LIN {X 0,Y 163.912,Z 823.88,A -85,B 0,C 180,E1 24592.6,E2 24592.6} C_VEL
LIN {X 0,Y 165.468,Z 824.667,A -85,B 0,C 180,E1 24598.513,E2 24598.513} C_VEL
LIN {X 0,Y 168.195,Z 823.745,A -85,B 0,C 180,E1 24603.972,E2 24603.972} C_VEL
LIN {X 0,Y 172.518,Z 820.86,A -85,B 0,C 180,E1 24609.607,E2 24609.607} C_VEL
LIN {X 0,Y 177.878,Z 816.328,A -85,B 0,C 180,E1 24614.638,E2 24614.638} C_VEL
LIN {X 0,Y 183.953,Z 810.223,A -85,B 0,C 180,E1 24619.07,E2 24619.07} C_VEL
LIN {X 0,Y 190.994,Z 802.117,A -85,B 0,C 180,E1 24623.221,E2 24623.221} C_VEL
LIN {X 0,Y 197.72,Z 793.266,A -85,B 0,C 180,E1 24626.552,E2 24626.552} C_VEL
LIN {X 0,Y 204.701,Z 782.624,A -85,B 0,C 180,E1 24629.553,E2 24629.553} C_VEL
LIN {X 0,Y 211.875,Z 769.936,A -85,B 0,C 180,E1 24632.25,E2 24632.25} C_VEL
LIN {X 0,Y 217.985,Z 757.04,A -85,B 0,C 180,E1 24634.33,E2 24634.33} C_VEL
LIN {X 0,Y 223.609,Z 742.371,A -85,B 0,C 180,E1 24636.121,E2 24636.121} C_VEL
LIN {X 0,Y 228.283,Z 726.827,A -85,B 0,C 180,E1 24637.541,E2 24637.541} C_VEL
LIN {X 0,Y 231.741,Z 710.644,A -85,B 0,C 180,E1 24638.599,E2 24638.599} C_VEL
LIN {X 0,Y 234.04,Z 693.375,A -85,B 0,C 180,E1 24639.347,E2 24639.347} C_VEL
LIN {X 0,Y 240.538,Z 622.169,A -85,B 0,C 180,E1 24641.299,E2 24641.299} C_VEL
LIN {X 0,Y 239.787,Z 607.797,A -85,B 0,C 180,E1 24642.742,E2 24642.742} C_VEL
LIN {X 0,Y 236.069,Z 599.284,A -85,B 0,C 180,E1 24645.591,E2 24645.591} C_VEL
LIN {X 0,Y 232.297,Z 591.41,A -85,B 0,C 180,E1 24649.02,E2 24649.02} C_VEL
LIN {X 0,Y 229.336,Z 585.624,A -85,B 0,C 180,E1 24652.358,E2 24652.358} C_VEL
LIN {X 0,Y 226.439,Z 580.103,A -85,B 0,C 180,E1 24656.962,E2 24656.962} C_VEL
LIN {X 0,Y 225.491,Z 578.392,A -85,B 0,C 180,E1 24659.237,E2 24659.237} C_VEL
LIN {X 0,Y 224.567,Z 575.979,A -85,B 0,C 180,E1 24664.596,E2 24664.596} C_VEL
LIN {X 0,Y 224.605,Z 575.941,A -85,B 0,C 180,E1 24665.938,E2 24665.938} C_VEL
LIN {X 0,Y 224.734,Z 577.003,A -85,B 0,C 180,E1 24667.755,E2 24667.755} C_VEL
LIN {X 0,Y 224.996,Z 580.824,A -85,B 0,C 180,E1 24670.283,E2 24670.283} C_VEL
LIN {X 0,Y 225.974,Z 586.453,A -85,B 0,C 180,E1 24673.585,E2 24673.585} C_VEL
LIN {X 0,Y 226.496,Z 587.496,A -85,B 0,C 180,E1 24674.544,E2 24674.544} C_VEL
LIN {X 0,Y 228.557,Z 590.668,A -85,B 0,C 180,E1 24677.509,E2 24677.509} C_VEL
LIN {X 0,Y 230.127,Z 593.107,A -85,B 0,C 180,E1 24679.347,E2 24679.347} C_VEL
LIN {X 0,Y 233.43,Z 598.617,A -85,B 0,C 180,E1 24682.541,E2 24682.541} C_VEL
LIN {X 0,Y 236.72,Z 604.703,A -85,B 0,C 180,E1 24685.252,E2 24685.252} C_VEL
LIN {X 0,Y 239.579,Z 610.555,A -85,B 0,C 180,E1 24687.307,E2 24687.307} C_VEL
LIN {X 0,Y 229.729,Z 717.254,A -85,B 0,C 180,E1 24690.022,E2 24690.022} C_VEL
LIN {X 0,Y 226.439,Z 735.292,A -85,B 0,C 180,E1 24690.738,E2 24690.738} C_VEL
LIN {X 0,Y 222.025,Z 751.667,A -85,B 0,C 180,E1 24691.665,E2 24691.665} C_VEL
LIN {X 0,Y 216.24,Z 768.025,A -85,B 0,C 180,E1 24692.942,E2 24692.942} C_VEL
LIN {X 0,Y 209.368,Z 783.676,A -85,B 0,C 180,E1 24694.631,E2 24694.631} C_VEL
LIN {X 0,Y 201.664,Z 798.456,A -85,B 0,C 180,E1 24696.802,E2 24696.802} C_VEL
LIN {X 0,Y 193.264,Z 812.488,A -85,B 0,C 180,E1 24699.57,E2 24699.57} C_VEL
LIN {X 0,Y 184.592,Z 825.393,A -85,B 0,C 180,E1 24703.01,E2 24703.01} C_VEL
LIN {X 0,Y 176.218,Z 836.632,A -85,B 0,C 180,E1 24707.088,E2 24707.088} C_VEL
LIN {X 0,Y 168.557,Z 846.394,A -85,B 0,C 180,E1 24711.909,E2 24711.909} C_VEL
LIN {X 0,Y 161.973,Z 854.666,A -85,B 0,C 180,E1 24717.518,E2 24717.518} C_VEL
LIN {X 0,Y 156.956,Z 861.39,A -85,B 0,C 180,E1 24723.925,E2 24723.925} C_VEL
LIN {X 0,Y 154.079,Z 866.16,A -85,B 0,C 180,E1 24730.674,E2 24730.674} C_VEL
LIN {X 0,Y 153.336,Z 869.27,A -85,B 0,C 180,E1 24737.986,E2 24737.986} C_VEL
LIN {X 0,Y 154.463,Z 870.381,A -85,B 0,C 180,E1 24744.801,E2 24744.801} C_VEL
LIN {X 0,Y 155.627,Z 870.068,A -85,B 0,C 180,E1 24749.264,E2 24749.264} C_VEL
LIN {X 0,Y 155.435,Z 869.168,A -85,B 0,C 180,E1 24752.213,E2 24752.213} C_VEL
LIN {X 0,Y 154.206,Z 866.135,A -85,B 0,C 180,E1 24757.826,E2 24757.826} C_VEL
LIN {X 0,Y 153.721,Z 861.161,A -85,B 0,C 180,E1 24763.926,E2 24763.926} C_VEL
LIN {X 0,Y 154.617,Z 854.342,A -85,B 0,C 180,E1 24770.044,E2 24770.044} C_VEL
LIN {X 0,Y 157.051,Z 845.493,A -85,B 0,C 180,E1 24776.059,E2 24776.059} C_VEL
LIN {X 0,Y 160.791,Z 835.076,A -85,B 0,C 180,E1 24781.49,E2 24781.49} C_VEL
LIN {X 0,Y 165.105,Z 824.003,A -85,B 0,C 180,E1 24785.975,E2 24785.975} C_VEL
LIN {X 0,Y 170.211,Z 811.051,A -85,B 0,C 180,E1 24790.034,E2 24790.034} C_VEL
LIN {X 0,Y 175.619,Z 796.472,A -85,B 0,C 180,E1 24793.544,E2 24793.544} C_VEL
LIN {X 0,Y 180.883,Z 780.858,A -85,B 0,C 180,E1 24796.397,E2 24796.397} C_VEL
LIN {X 0,Y 185.452,Z 765.246,A -85,B 0,C 180,E1 24798.54,E2 24798.54} C_VEL
LIN {X 0,Y 189.399,Z 748.752,A -85,B 0,C 180,E1 24800.199,E2 24800.199} C_VEL
LIN {X 0,Y 192.481,Z 731.114,A -85,B 0,C 180,E1 24801.451,E2 24801.451} C_VEL
LIN {X 0,Y 194.415,Z 712.665,A -85,B 0,C 180,E1 24802.3,E2 24802.3} C_VEL
LIN {X 0,Y 202.526,Z 587.616,A -85,B 0,C 180,E1 24806.166,E2 24806.166} C_VEL
LIN {X 0,Y 202.127,Z 580.747,A -85,B 0,C 180,E1 24806.612,E2 24806.612} C_VEL
LIN {X 0,Y 194.488,Z 565.099,A -85,B 0,C 180,E1 24809.663,E2 24809.663} C_VEL
LIN {X 0,Y 186.875,Z 551.393,A -85,B 0,C 180,E1 24813.036,E2 24813.036} C_VEL
LIN {X 0,Y 183.387,Z 545.505,A -85,B 0,C 180,E1 24814.833,E2 24814.833} C_VEL
LIN {X 0,Y 180.867,Z 537.663,A -85,B 0,C 180,E1 24819.281,E2 24819.281} C_VEL
LIN {X 0,Y 178.385,Z 530.763,A -85,B 0,C 180,E1 24824.06,E2 24824.06} C_VEL
LIN {X 0,Y 176.409,Z 525.313,A -85,B 0,C 180,E1 24828.559,E2 24828.559} C_VEL
LIN {X 0,Y 174.729,Z 521.276,A -85,B 0,C 180,E1 24832.768,E2 24832.768} C_VEL
LIN {X 0,Y 173.264,Z 517.729,A -85,B 0,C 180,E1 24837.355,E2 24837.355} C_VEL
LIN {X 0,Y 171.645,Z 513.857,A -85,B 0,C 180,E1 24845.013,E2 24845.013} C_VEL
LIN {X 0,Y 170.767,Z 512.763,A -85,B 0,C 180,E1 24851.484,E2 24851.484} C_VEL
LIN {X 0,Y 170.898,Z 512.989,A -85,B 0,C 180,E1 24858.065,E2 24858.065} C_VEL
LIN {X 0,Y 171.446,Z 514.088,A -85,B 0,C 180,E1 24862.639,E2 24862.639} C_VEL
LIN {X 0,Y 172.787,Z 517.698,A -85,B 0,C 180,E1 24869.846,E2 24869.846} C_VEL
LIN {X 0,Y 174.086,Z 521.491,A -85,B 0,C 180,E1 24874.782,E2 24874.782} C_VEL
LIN {X 0,Y 175.487,Z 525.746,A -85,B 0,C 180,E1 24879.205,E2 24879.205} C_VEL
LIN {X 0,Y 177.274,Z 531.253,A -85,B 0,C 180,E1 24883.928,E2 24883.928} C_VEL
LIN {X 0,Y 179.348,Z 538.517,A -85,B 0,C 180,E1 24889.062,E2 24889.062} C_VEL
LIN {X 0,Y 181.315,Z 546.515,A -85,B 0,C 180,E1 24893.839,E2 24893.839} C_VEL
LIN {X 0,Y 182.26,Z 550.218,A -85,B 0,C 180,E1 24895.653,E2 24895.653} C_VEL
LIN {X 0,Y 188.742,Z 562.541,A -85,B 0,C 180,E1 24898.821,E2 24898.821} C_VEL
LIN {X 0,Y 194.269,Z 574.356,A -85,B 0,C 180,E1 24901.293,E2 24901.293} C_VEL
LIN {X 0,Y 197.448,Z 613.753,A -85,B 0,C 180,E1 24904.282,E2 24904.282} C_VEL
LIN {X 0,Y 191.617,Z 696.457,A -85,B 0,C 180,E1 24907.072,E2 24907.072} C_VEL
LIN {X 0,Y 189.522,Z 713.957,A -85,B 0,C 180,E1 24908.201,E2 24908.201} C_VEL
LIN {X 0,Y 186.823,Z 729.138,A -85,B 0,C 180,E1 24909.642,E2 24909.642} C_VEL
LIN {X 0,Y 183.113,Z 744.763,A -85,B 0,C 180,E1 24911.701,E2 24911.701} C_VEL
LIN {X 0,Y 178.862,Z 759.406,A -85,B 0,C 180,E1 24914.268,E2 24914.268} C_VEL
LIN {X 0,Y 174.27,Z 772.863,A -85,B 0,C 180,E1 24917.407,E2 24917.407} C_VEL
LIN {X 0,Y 169.559,Z 785.286,A -85,B 0,C 180,E1 24921.18,E2 24921.18} C_VEL
LIN {X 0,Y 165.156,Z 796.018,A -85,B 0,C 180,E1 24925.485,E2 24925.485} C_VEL
LIN {X 0,Y 161.321,Z 805.271,A -85,B 0,C 180,E1 24930.354,E2 24930.354} C_VEL
LIN {X 0,Y 158.455,Z 812.493,A -85,B 0,C 180,E1 24935.431,E2 24935.431} C_VEL
LIN {X 0,Y 156.409,Z 818.667,A -85,B 0,C 180,E1 24941.429,E2 24941.429} C_VEL
LIN {X 0,Y 155.668,Z 822.689,A -85,B 0,C 180,E1 24947.184,E2 24947.184} C_VEL
LIN {X 0,Y 156.104,Z 825.148,A -85,B 0,C 180,E1 24953.397,E2 24953.397} C_VEL
LIN {X 0,Y 157.914,Z 825.868,A -85,B 0,C 180,E1 24959.595,E2 24959.595} C_VEL
LIN {X 0,Y 161.208,Z 824.71,A -85,B 0,C 180,E1 24965.662,E2 24965.662} C_VEL
LIN {X 0,Y 166.048,Z 821.661,A -85,B 0,C 180,E1 24971.48,E2 24971.48} C_VEL
LIN {X 0,Y 171.989,Z 816.833,A -85,B 0,C 180,E1 24976.685,E2 24976.685} C_VEL
LIN {X 0,Y 179.003,Z 810.086,A -85,B 0,C 180,E1 24981.443,E2 24981.443} C_VEL
LIN {X 0,Y 186.039,Z 802.321,A -85,B 0,C 180,E1 24985.314,E2 24985.314} C_VEL
LIN {X 0,Y 193.796,Z 792.352,A -85,B 0,C 180,E1 24988.919,E2 24988.919} C_VEL
LIN {X 0,Y 201.556,Z 780.804,A -85,B 0,C 180,E1 24992.006,E2 24992.006} C_VEL
LIN {X 0,Y 208.433,Z 768.711,A -85,B 0,C 180,E1 24994.422,E2 24994.422} C_VEL
LIN {X 0,Y 215.191,Z 754.374,A -85,B 0,C 180,E1 24996.585,E2 24996.585} C_VEL
LIN {X 0,Y 220.706,Z 739.879,A -85,B 0,C 180,E1 24998.233,E2 24998.233} C_VEL
LIN {X 0,Y 225.369,Z 723.672,A -85,B 0,C 180,E1 24999.588,E2 24999.588} C_VEL
LIN {X 0,Y 228.761,Z 706.983,A -85,B 0,C 180,E1 25000.578,E2 25000.578} C_VEL
LIN {X 0,Y 230.892,Z 688.612,A -85,B 0,C 180,E1 25001.264,E2 25001.264} C_VEL
LIN {X 0,Y 237.023,Z 623.672,A -85,B 0,C 180,E1 25003.014,E2 25003.014} C_VEL
LIN {X 0,Y 236.583,Z 612.854,A -85,B 0,C 180,E1 25004.118,E2 25004.118} C_VEL
LIN {X 0,Y 233.097,Z 604.36,A -85,B 0,C 180,E1 25007.111,E2 25007.111} C_VEL
LIN {X 0,Y 230.024,Z 597.815,A -85,B 0,C 180,E1 25010.176,E2 25010.176} C_VEL
LIN {X 0,Y 227.629,Z 592.775,A -85,B 0,C 180,E1 25013.188,E2 25013.188} C_VEL
LIN {X 0,Y 224.989,Z 587.376,A -85,B 0,C 180,E1 25017.835,E2 25017.835} C_VEL
LIN {X 0,Y 223.577,Z 584.108,A -85,B 0,C 180,E1 25023.846,E2 25023.846} C_VEL
LIN {X 0,Y 223.986,Z 584.134,A -85,B 0,C 180,E1 25028.471,E2 25028.471} C_VEL
LIN {X 0,Y 224.955,Z 585.243,A -85,B 0,C 180,E1 25031.537,E2 25031.537} C_VEL
LIN {X 0,Y 226.496,Z 587.496,A -85,B 0,C 180,E1 25034.544,E2 25034.544} C_VEL
LIN {X 0,Y 227.426,Z 589.736,A -85,B 0,C 180,E1 25036.103,E2 25036.103} C_VEL
LIN {X 0,Y 228.666,Z 595.152,A -85,B 0,C 180,E1 25038.205,E2 25038.205} C_VEL
LIN {X 0,Y 231,Z 604.636,A -85,B 0,C 180,E1 25041.335,E2 25041.335} C_VEL
LIN {X 0,Y 231.718,Z 606.293,A -85,B 0,C 180,E1 25042.049,E2 25042.049} C_VEL
LIN {X 0,Y 234.684,Z 612.043,A -85,B 0,C 180,E1 25044.611,E2 25044.611} C_VEL
LIN {X 0,Y 235.967,Z 614.984,A -85,B 0,C 180,E1 25045.643,E2 25045.643} C_VEL
LIN {X 0,Y 226.245,Z 716.589,A -85,B 0,C 180,E1 25048.199,E2 25048.199} C_VEL
LIN {X 0,Y 222.849,Z 734.651,A -85,B 0,C 180,E1 25048.9,E2 25048.9} C_VEL
LIN {X 0,Y 218.339,Z 750.91,A -85,B 0,C 180,E1 25049.798,E2 25049.798} C_VEL
LIN {X 0,Y 212.387,Z 767.251,A -85,B 0,C 180,E1 25051.041,E2 25051.041} C_VEL
LIN {X 0,Y 205.441,Z 782.574,A -85,B 0,C 180,E1 25052.652,E2 25052.652} C_VEL
LIN {X 0,Y 197.661,Z 797.012,A -85,B 0,C 180,E1 25054.716,E2 25054.716} C_VEL
LIN {X 0,Y 188.883,Z 811.075,A -85,B 0,C 180,E1 25057.437,E2 25057.437} C_VEL
LIN {X 0,Y 180.383,Z 823.142,A -85,B 0,C 180,E1 25060.59,E2 25060.59} C_VEL
LIN {X 0,Y 171.44,Z 834.634,A -85,B 0,C 180,E1 25064.642,E2 25064.642} C_VEL
LIN {X 0,Y 163.116,Z 844.539,A -85,B 0,C 180,E1 25069.478,E2 25069.478} C_VEL
LIN {X 0,Y 155.777,Z 853.017,A -85,B 0,C 180,E1 25075.241,E2 25075.241} C_VEL
LIN {X 0,Y 150.108,Z 859.783,A -85,B 0,C 180,E1 25081.776,E2 25081.776} C_VEL
LIN {X 0,Y 146.61,Z 864.678,A -85,B 0,C 180,E1 25088.811,E2 25088.811} C_VEL
LIN {X 0,Y 145.355,Z 867.881,A -85,B 0,C 180,E1 25096.475,E2 25096.475} C_VEL
LIN {X 0,Y 146.249,Z 869.12,A -85,B 0,C 180,E1 25103.721,E2 25103.721} C_VEL
LIN {X 0,Y 147.713,Z 868.776,A -85,B 0,C 180,E1 25109.225,E2 25109.225} C_VEL
LIN {X 0,Y 147.462,Z 867.817,A -85,B 0,C 180,E1 25112.332,E2 25112.332} C_VEL
LIN {X 0,Y 146.186,Z 864.662,A -85,B 0,C 180,E1 25118.259,E2 25118.259} C_VEL
LIN {X 0,Y 145.801,Z 859.479,A -85,B 0,C 180,E1 25124.777,E2 25124.777} C_VEL
LIN {X 0,Y 147.037,Z 852.093,A -85,B 0,C 180,E1 25131.544,E2 25131.544} C_VEL
LIN {X 0,Y 149.911,Z 842.967,A -85,B 0,C 180,E1 25137.833,E2 25137.833} C_VEL
LIN {X 0,Y 153.798,Z 832.968,A -85,B 0,C 180,E1 25143.1,E2 25143.1} C_VEL
LIN {X 0,Y 158.628,Z 821.261,A -85,B 0,C 180,E1 25147.856,E2 25147.856} C_VEL
LIN {X 0,Y 164.2,Z 807.761,A -85,B 0,C 180,E1 25152.054,E2 25152.054} C_VEL
LIN {X 0,Y 169.836,Z 793.102,A -85,B 0,C 180,E1 25155.527,E2 25155.527} C_VEL
LIN {X 0,Y 175.01,Z 778.109,A -85,B 0,C 180,E1 25158.209,E2 25158.209} C_VEL
LIN {X 0,Y 179.796,Z 761.819,A -85,B 0,C 180,E1 25160.373,E2 25160.373} C_VEL
LIN {X 0,Y 183.906,Z 744.505,A -85,B 0,C 180,E1 25162.031,E2 25162.031} C_VEL
LIN {X 0,Y 186.876,Z 726.688,A -85,B 0,C 180,E1 25163.227,E2 25163.227} C_VEL
LIN {X 0,Y 188.636,Z 708.081,A -85,B 0,C 180,E1 25164.002,E2 25164.002} C_VEL
LIN {X 0,Y 196.745,Z 588.477,A -85,B 0,C 180,E1 25167.739,E2 25167.739} C_VEL
LIN {X 0,Y 196.482,Z 584.015,A -85,B 0,C 180,E1 25168.047,E2 25168.047} C_VEL
LIN {X 0,Y 189.501,Z 569.514,A -85,B 0,C 180,E1 25171.047,E2 25171.047} C_VEL
LIN {X 0,Y 182.65,Z 556.895,A -85,B 0,C 180,E1 25174.29,E2 25174.29} C_VEL
LIN {X 0,Y 175.931,Z 545.772,A -85,B 0,C 180,E1 25177.97,E2 25177.97} C_VEL
LIN {X 0,Y 173.293,Z 537.692,A -85,B 0,C 180,E1 25183.293,E2 25183.293} C_VEL
LIN {X 0,Y 170.883,Z 531.024,A -85,B 0,C 180,E1 25188.868,E2 25188.868} C_VEL
LIN {X 0,Y 169.257,Z 526.989,A -85,B 0,C 180,E1 25193.215,E2 25193.215} C_VEL
LIN {X 0,Y 167.952,Z 523.675,A -85,B 0,C 180,E1 25197.612,E2 25197.612} C_VEL
LIN {X 0,Y 166.457,Z 519.94,A -85,B 0,C 180,E1 25205.17,E2 25205.17} C_VEL
LIN {X 0,Y 165.605,Z 518.873,A -85,B 0,C 180,E1 25211.847,E2 25211.847} C_VEL
LIN {X 0,Y 165.788,Z 519.189,A -85,B 0,C 180,E1 25218.761,E2 25218.761} C_VEL
LIN {X 0,Y 166.206,Z 520.189,A -85,B 0,C 180,E1 25222.645,E2 25222.645} C_VEL
LIN {X 0,Y 167.387,Z 523.662,A -85,B 0,C 180,E1 25229.722,E2 25229.722} C_VEL
LIN {X 0,Y 168.576,Z 527.414,A -85,B 0,C 180,E1 25234.709,E2 25234.709} C_VEL
LIN {X 0,Y 169.863,Z 531.465,A -85,B 0,C 180,E1 25239.039,E2 25239.039} C_VEL
LIN {X 0,Y 171.533,Z 537.047,A -85,B 0,C 180,E1 25243.92,E2 25243.92} C_VEL
LIN {X 0,Y 173.338,Z 543.924,A -85,B 0,C 180,E1 25248.883,E2 25248.883} C_VEL
LIN {X 0,Y 174.89,Z 549.948,A -85,B 0,C 180,E1 25252.478,E2 25252.478} C_VEL
LIN {X 0,Y 181.396,Z 561.8,A -85,B 0,C 180,E1 25256.055,E2 25256.055} C_VEL
LIN {X 0,Y 188.043,Z 575.718,A -85,B 0,C 180,E1 25259.339,E2 25259.339} C_VEL
LIN {X 0,Y 189.015,Z 578.721,A -85,B 0,C 180,E1 25259.841,E2 25259.841} C_VEL
LIN {X 0,Y 191.643,Z 614.777,A -85,B 0,C 180,E1 25262.669,E2 25262.669} C_VEL
LIN {X 0,Y 185.611,Z 696.897,A -85,B 0,C 180,E1 25265.472,E2 25265.472} C_VEL
LIN {X 0,Y 183.431,Z 714.382,A -85,B 0,C 180,E1 25266.613,E2 25266.613} C_VEL
LIN {X 0,Y 180.378,Z 730.668,A -85,B 0,C 180,E1 25268.198,E2 25268.198} C_VEL
LIN {X 0,Y 176.504,Z 746.135,A -85,B 0,C 180,E1 25270.302,E2 25270.302} C_VEL
LIN {X 0,Y 172.059,Z 760.666,A -85,B 0,C 180,E1 25272.934,E2 25272.934} C_VEL
LIN {X 0,Y 167.069,Z 774.537,A -85,B 0,C 180,E1 25276.298,E2 25276.298} C_VEL
LIN {X 0,Y 162.309,Z 786.438,A -85,B 0,C 180,E1 25280.067,E2 25280.067} C_VEL
LIN {X 0,Y 157.681,Z 797.143,A -85,B 0,C 180,E1 25284.541,E2 25284.541} C_VEL
LIN {X 0,Y 153.643,Z 806.389,A -85,B 0,C 180,E1 25289.626,E2 25289.626} C_VEL
LIN {X 0,Y 150.57,Z 813.743,A -85,B 0,C 180,E1 25295.07,E2 25295.07} C_VEL
LIN {X 0,Y 148.482,Z 819.793,A -85,B 0,C 180,E1 25301.261,E2 25301.261} C_VEL
LIN {X 0,Y 147.729,Z 823.861,A -85,B 0,C 180,E1 25307.382,E2 25307.382} C_VEL
LIN {X 0,Y 148.248,Z 826.317,A -85,B 0,C 180,E1 25313.87,E2 25313.87} C_VEL
LIN {X 0,Y 150.241,Z 827.064,A -85,B 0,C 180,E1 25320.383,E2 25320.383} C_VEL
LIN {X 0,Y 153.817,Z 825.948,A -85,B 0,C 180,E1 25326.728,E2 25326.728} C_VEL
LIN {X 0,Y 159.009,Z 822.939,A -85,B 0,C 180,E1 25332.773,E2 25332.773} C_VEL
LIN {X 0,Y 165.266,Z 818.258,A -85,B 0,C 180,E1 25338.085,E2 25338.085} C_VEL
LIN {X 0,Y 172.752,Z 811.533,A -85,B 0,C 180,E1 25343.007,E2 25343.007} C_VEL
LIN {X 0,Y 180.542,Z 803.433,A -85,B 0,C 180,E1 25347.129,E2 25347.129} C_VEL
LIN {X 0,Y 188.261,Z 794.047,A -85,B 0,C 180,E1 25350.575,E2 25350.575} C_VEL
LIN {X 0,Y 196.467,Z 782.447,A -85,B 0,C 180,E1 25353.719,E2 25353.719} C_VEL
LIN {X 0,Y 203.817,Z 770.182,A -85,B 0,C 180,E1 25356.191,E2 25356.191} C_VEL
LIN {X 0,Y 210.554,Z 756.575,A -85,B 0,C 180,E1 25358.259,E2 25358.259} C_VEL
LIN {X 0,Y 216.601,Z 741.506,A -85,B 0,C 180,E1 25359.986,E2 25359.986} C_VEL
LIN {X 0,Y 221.327,Z 726.055,A -85,B 0,C 180,E1 25361.291,E2 25361.291} C_VEL
LIN {X 0,Y 225.032,Z 708.952,A -85,B 0,C 180,E1 25362.322,E2 25362.322} C_VEL
LIN {X 0,Y 227.239,Z 691.89,A -85,B 0,C 180,E1 25362.988,E2 25362.988} C_VEL
LIN {X 0,Y 233.751,Z 625.32,A -85,B 0,C 180,E1 25364.77,E2 25364.77} C_VEL
LIN {X 0,Y 233.536,Z 617.898,A -85,B 0,C 180,E1 25365.558,E2 25365.558} C_VEL
LIN {X 0,Y 230.437,Z 610.119,A -85,B 0,C 180,E1 25368.486,E2 25368.486} C_VEL
LIN {X 0,Y 228.06,Z 604.663,A -85,B 0,C 180,E1 25371.109,E2 25371.109} C_VEL
LIN {X 0,Y 226.04,Z 600.109,A -85,B 0,C 180,E1 25373.905,E2 25373.905} C_VEL
LIN {X 0,Y 223.704,Z 594.913,A -85,B 0,C 180,E1 25378.463,E2 25378.463} C_VEL
LIN {X 0,Y 222.524,Z 591.829,A -85,B 0,C 180,E1 25384.897,E2 25384.897} C_VEL
LIN {X 0,Y 223.496,Z 592.511,A -85,B 0,C 180,E1 25390.308,E2 25390.308} C_VEL
LIN {X 0,Y 225.907,Z 596.185,A -85,B 0,C 180,E1 25395.268,E2 25395.268} C_VEL
LIN {X 0,Y 228.493,Z 600.587,A -85,B 0,C 180,E1 25398.761,E2 25398.761} C_VEL
LIN {X 0,Y 231.464,Z 605.781,A -85,B 0,C 180,E1 25401.807,E2 25401.807} C_VEL
LIN {X 0,Y 231.718,Z 606.293,A -85,B 0,C 180,E1 25402.049,E2 25402.049} C_VEL
LIN {X 0,Y 232.472,Z 608.94,A -85,B 0,C 180,E1 25402.851,E2 25402.851} C_VEL
LIN {X 0,Y 232.864,Z 613.541,A -85,B 0,C 180,E1 25403.552,E2 25403.552} C_VEL
LIN {X 0,Y 232.713,Z 619.941,A -85,B 0,C 180,E1 25404.032,E2 25404.032} C_VEL
LIN {X 0,Y 231.331,Z 633.276,A -85,B 0,C 180,E1 25404.316,E2 25404.316} C_VEL
LIN {X 0,Y 230.508,Z 640.63,A -85,B 0,C 180,E1 25404.432,E2 25404.432} C_VEL
LIN {X 0,Y 222.986,Z 715.998,A -85,B 0,C 180,E1 25406.324,E2 25406.324} C_VEL
LIN {X 0,Y 219.471,Z 734.121,A -85,B 0,C 180,E1 25407.009,E2 25407.009} C_VEL
LIN {X 0,Y 214.484,Z 751.431,A -85,B 0,C 180,E1 25407.947,E2 25407.947} C_VEL
LIN {X 0,Y 208.371,Z 767.413,A -85,B 0,C 180,E1 25409.154,E2 25409.154} C_VEL
LIN {X 0,Y 200.829,Z 783.246,A -85,B 0,C 180,E1 25410.817,E2 25410.817} C_VEL
LIN {X 0,Y 192.436,Z 798.023,A -85,B 0,C 180,E1 25412.953,E2 25412.953} C_VEL
LIN {X 0,Y 183.369,Z 811.76,A -85,B 0,C 180,E1 25415.665,E2 25415.665} C_VEL
LIN {X 0,Y 173.893,Z 824.307,A -85,B 0,C 180,E1 25419.084,E2 25419.084} C_VEL
LIN {X 0,Y 164.626,Z 835.315,A -85,B 0,C 180,E1 25423.213,E2 25423.213} C_VEL
LIN {X 0,Y 155.968,Z 844.875,A -85,B 0,C 180,E1 25428.187,E2 25428.187} C_VEL
LIN {X 0,Y 148.367,Z 852.971,A -85,B 0,C 180,E1 25434.106,E2 25434.106} C_VEL
LIN {X 0,Y 142.357,Z 859.436,A -85,B 0,C 180,E1 25441.013,E2 25441.013} C_VEL
LIN {X 0,Y 138.558,Z 864.229,A -85,B 0,C 180,E1 25448.851,E2 25448.851} C_VEL
LIN {X 0,Y 137.409,Z 866.96,A -85,B 0,C 180,E1 25456.536,E2 25456.536} C_VEL
LIN {X 0,Y 138.415,Z 867.935,A -85,B 0,C 180,E1 25464.196,E2 25464.196} C_VEL
LIN {X 0,Y 139.869,Z 867.395,A -85,B 0,C 180,E1 25469.591,E2 25469.591} C_VEL
LIN {X 0,Y 139.374,Z 866.29,A -85,B 0,C 180,E1 25472.879,E2 25472.879} C_VEL
LIN {X 0,Y 138.053,Z 862.621,A -85,B 0,C 180,E1 25479.59,E2 25479.59} C_VEL
LIN {X 0,Y 137.971,Z 857.167,A -85,B 0,C 180,E1 25486.418,E2 25486.418} C_VEL
LIN {X 0,Y 139.556,Z 849.842,A -85,B 0,C 180,E1 25493.208,E2 25493.208} C_VEL
LIN {X 0,Y 142.66,Z 841.003,A -85,B 0,C 180,E1 25499.381,E2 25499.381} C_VEL
LIN {X 0,Y 146.936,Z 830.745,A -85,B 0,C 180,E1 25504.863,E2 25504.863} C_VEL
LIN {X 0,Y 152.47,Z 818.152,A -85,B 0,C 180,E1 25509.991,E2 25509.991} C_VEL
LIN {X 0,Y 158.153,Z 804.976,A -85,B 0,C 180,E1 25514.062,E2 25514.062} C_VEL
LIN {X 0,Y 163.731,Z 790.988,A -85,B 0,C 180,E1 25517.355,E2 25517.355} C_VEL
LIN {X 0,Y 169.323,Z 775.129,A -85,B 0,C 180,E1 25520.145,E2 25520.145} C_VEL
LIN {X 0,Y 174.345,Z 758.297,A -85,B 0,C 180,E1 25522.32,E2 25522.32} C_VEL
LIN {X 0,Y 178.291,Z 741.664,A -85,B 0,C 180,E1 25523.859,E2 25523.859} C_VEL
LIN {X 0,Y 181.17,Z 723.955,A -85,B 0,C 180,E1 25525.001,E2 25525.001} C_VEL
LIN {X 0,Y 183.039,Z 702.995,A -85,B 0,C 180,E1 25525.816,E2 25525.816} C_VEL
LIN {X 0,Y 191.118,Z 589.134,A -85,B 0,C 180,E1 25529.418,E2 25529.418} C_VEL
LIN {X 0,Y 190.825,Z 587.022,A -85,B 0,C 180,E1 25529.628,E2 25529.628} C_VEL
LIN {X 0,Y 183.757,Z 572.094,A -85,B 0,C 180,E1 25532.934,E2 25532.934} C_VEL
LIN {X 0,Y 176.814,Z 559.558,A -85,B 0,C 180,E1 25536.506,E2 25536.506} C_VEL
LIN {X 0,Y 171.109,Z 550.361,A -85,B 0,C 180,E1 25539.833,E2 25539.833} C_VEL
LIN {X 0,Y 168.394,Z 545.783,A -85,B 0,C 180,E1 25541.811,E2 25541.811} C_VEL
LIN {X 0,Y 166.095,Z 539.006,A -85,B 0,C 180,E1 25547.131,E2 25547.131} C_VEL
LIN {X 0,Y 164.208,Z 533.463,A -85,B 0,C 180,E1 25552.654,E2 25552.654} C_VEL
LIN {X 0,Y 162.647,Z 529.623,A -85,B 0,C 180,E1 25557.887,E2 25557.887} C_VEL
LIN {X 0,Y 161.268,Z 526.02,A -85,B 0,C 180,E1 25565.337,E2 25565.337} C_VEL
LIN {X 0,Y 160.459,Z 524.995,A -85,B 0,C 180,E1 25571.953,E2 25571.953} C_VEL
LIN {X 0,Y 160.616,Z 525.304,A -85,B 0,C 180,E1 25578.888,E2 25578.888} C_VEL
LIN {X 0,Y 160.965,Z 526.301,A -85,B 0,C 180,E1 25582.652,E2 25582.652} C_VEL
LIN {X 0,Y 162.005,Z 529.638,A -85,B 0,C 180,E1 25589.588,E2 25589.588} C_VEL
LIN {X 0,Y 163.019,Z 533.087,A -85,B 0,C 180,E1 25594.353,E2 25594.353} C_VEL
LIN {X 0,Y 164.236,Z 537.157,A -85,B 0,C 180,E1 25598.834,E2 25598.834} C_VEL
LIN {X 0,Y 165.795,Z 542.824,A -85,B 0,C 180,E1 25603.911,E2 25603.911} C_VEL
LIN {X 0,Y 167.577,Z 549.695,A -85,B 0,C 180,E1 25608.763,E2 25608.763} C_VEL
LIN {X 0,Y 172.346,Z 558.116,A -85,B 0,C 180,E1 25611.891,E2 25611.891} C_VEL
LIN {X 0,Y 177.4,Z 567.568,A -85,B 0,C 180,E1 25614.811,E2 25614.811} C_VEL
LIN {X 0,Y 183.615,Z 581.049,A -85,B 0,C 180,E1 25618.083,E2 25618.083} C_VEL
LIN {X 0,Y 186.031,Z 615.401,A -85,B 0,C 180,E1 25620.944,E2 25620.944} C_VEL
LIN {X 0,Y 179.743,Z 697.491,A -85,B 0,C 180,E1 25623.775,E2 25623.775} C_VEL
LIN {X 0,Y 177.472,Z 714.924,A -85,B 0,C 180,E1 25624.926,E2 25624.926} C_VEL
LIN {X 0,Y 174.334,Z 731.038,A -85,B 0,C 180,E1 25626.508,E2 25626.508} C_VEL
LIN {X 0,Y 170.274,Z 746.591,A -85,B 0,C 180,E1 25628.649,E2 25628.649} C_VEL
LIN {X 0,Y 165.61,Z 761.209,A -85,B 0,C 180,E1 25631.337,E2 25631.337} C_VEL
LIN {X 0,Y 160.55,Z 774.671,A -85,B 0,C 180,E1 25634.652,E2 25634.652} C_VEL
LIN {X 0,Y 155.532,Z 786.639,A -85,B 0,C 180,E1 25638.504,E2 25638.504} C_VEL
LIN {X 0,Y 150.949,Z 796.795,A -85,B 0,C 180,E1 25642.769,E2 25642.769} C_VEL
LIN {X 0,Y 146.534,Z 806.293,A -85,B 0,C 180,E1 25648.044,E2 25648.044} C_VEL
LIN {X 0,Y 143,Z 814.284,A -85,B 0,C 180,E1 25654.009,E2 25654.009} C_VEL
LIN {X 0,Y 140.756,Z 820.247,A -85,B 0,C 180,E1 25660.229,E2 25660.229} C_VEL
LIN {X 0,Y 139.802,Z 824.749,A -85,B 0,C 180,E1 25667.051,E2 25667.051} C_VEL
LIN {X 0,Y 140.319,Z 827.384,A -85,B 0,C 180,E1 25673.963,E2 25673.963} C_VEL
LIN {X 0,Y 142.557,Z 828.257,A -85,B 0,C 180,E1 25681.164,E2 25681.164} C_VEL
LIN {X 0,Y 146.199,Z 827.328,A -85,B 0,C 180,E1 25687.501,E2 25687.501} C_VEL
LIN {X 0,Y 151.666,Z 824.474,A -85,B 0,C 180,E1 25693.805,E2 25693.805} C_VEL
LIN {X 0,Y 158.459,Z 819.843,A -85,B 0,C 180,E1 25699.464,E2 25699.464} C_VEL
LIN {X 0,Y 166.077,Z 813.497,A -85,B 0,C 180,E1 25704.365,E2 25704.365} C_VEL
LIN {X 0,Y 174.405,Z 805.398,A -85,B 0,C 180,E1 25708.672,E2 25708.672} C_VEL
LIN {X 0,Y 182.802,Z 795.853,A -85,B 0,C 180,E1 25712.294,E2 25712.294} C_VEL
LIN {X 0,Y 191.294,Z 784.474,A -85,B 0,C 180,E1 25715.43,E2 25715.43} C_VEL
LIN {X 0,Y 199.051,Z 772.248,A -85,B 0,C 180,E1 25717.935,E2 25717.935} C_VEL
LIN {X 0,Y 205.942,Z 759.149,A -85,B 0,C 180,E1 25719.958,E2 25719.958} C_VEL
LIN {X 0,Y 212.372,Z 744.047,A -85,B 0,C 180,E1 25721.714,E2 25721.714} C_VEL
LIN {X 0,Y 217.431,Z 728.801,A -85,B 0,C 180,E1 25723.035,E2 25723.035} C_VEL
LIN {X 0,Y 221.294,Z 712.442,A -85,B 0,C 180,E1 25724.052,E2 25724.052} C_VEL
LIN {X 0,Y 223.86,Z 695.119,A -85,B 0,C 180,E1 25724.771,E2 25724.771} C_VEL
LIN {X 0,Y 230.753,Z 626.94,A -85,B 0,C 180,E1 25726.579,E2 25726.579} C_VEL
LIN {X 0,Y 230.651,Z 622.932,A -85,B 0,C 180,E1 25727.036,E2 25727.036} C_VEL
LIN {X 0,Y 228.085,Z 616.24,A -85,B 0,C 180,E1 25729.709,E2 25729.709} C_VEL
LIN {X 0,Y 226.091,Z 611.343,A -85,B 0,C 180,E1 25732.184,E2 25732.184} C_VEL
LIN {X 0,Y 224.482,Z 607.474,A -85,B 0,C 180,E1 25734.632,E2 25734.632} C_VEL
LIN {X 0,Y 222.445,Z 602.456,A -85,B 0,C 180,E1 25739.098,E2 25739.098} C_VEL
LIN {X 0,Y 221.503,Z 599.763,A -85,B 0,C 180,E1 25744.92,E2 25744.92} C_VEL
LIN {X 0,Y 222.399,Z 600.398,A -85,B 0,C 180,E1 25750.098,E2 25750.098} C_VEL
LIN {X 0,Y 224.571,Z 603.904,A -85,B 0,C 180,E1 25754.833,E2 25754.833} C_VEL
LIN {X 0,Y 226.9,Z 608.068,A -85,B 0,C 180,E1 25758.165,E2 25758.165} C_VEL
LIN {X 0,Y 229.596,Z 613.074,A -85,B 0,C 180,E1 25761.122,E2 25761.122} C_VEL
LIN {X 0,Y 232.538,Z 619.088,A -85,B 0,C 180,E1 25763.839,E2 25763.839} C_VEL
LIN {X 0,Y 232.558,Z 620.037,A -85,B 0,C 180,E1 25763.938,E2 25763.938} C_VEL
LIN {X 0,Y 230.508,Z 640.63,A -85,B 0,C 180,E1 25764.432,E2 25764.432} C_VEL
LIN {X 0,Y 229.395,Z 648.312,A -85,B 0,C 180,E1 25764.388,E2 25764.388} C_VEL
LIN {X 0,Y 225.185,Z 668.771,A -85,B 0,C 180,E1 25763.406,E2 25763.406} C_VEL
LIN {X 0,Y 224.262,Z 675.367,A -85,B 0,C 180,E1 25763.38,E2 25763.38} C_VEL
LIN {X 0,Y 219.965,Z 715.881,A -85,B 0,C 180,E1 25764.403,E2 25764.403} C_VEL
LIN {X 0,Y 216.212,Z 734.333,A -85,B 0,C 180,E1 25765.088,E2 25765.088} C_VEL
LIN {X 0,Y 211.282,Z 750.784,A -85,B 0,C 180,E1 25765.955,E2 25765.955} C_VEL
LIN {X 0,Y 205.007,Z 766.668,A -85,B 0,C 180,E1 25767.116,E2 25767.116} C_VEL
LIN {X 0,Y 197.238,Z 782.44,A -85,B 0,C 180,E1 25768.72,E2 25768.72} C_VEL
LIN {X 0,Y 188.558,Z 797.192,A -85,B 0,C 180,E1 25770.793,E2 25770.793} C_VEL
LIN {X 0,Y 179.135,Z 810.897,A -85,B 0,C 180,E1 25773.443,E2 25773.443} C_VEL
LIN {X 0,Y 169.563,Z 822.999,A -85,B 0,C 180,E1 25776.684,E2 25776.684} C_VEL
LIN {X 0,Y 159.766,Z 834.038,A -85,B 0,C 180,E1 25780.778,E2 25780.778} C_VEL
LIN {X 0,Y 150.488,Z 843.604,A -85,B 0,C 180,E1 25785.763,E2 25785.763} C_VEL
LIN {X 0,Y 142.223,Z 851.692,A -85,B 0,C 180,E1 25791.783,E2 25791.783} C_VEL
LIN {X 0,Y 135.524,Z 858.164,A -85,B 0,C 180,E1 25798.907,E2 25798.907} C_VEL
LIN {X 0,Y 131.087,Z 862.964,A -85,B 0,C 180,E1 25807.109,E2 25807.109} C_VEL
LIN {X 0,Y 129.473,Z 865.813,A -85,B 0,C 180,E1 25815.694,E2 25815.694} C_VEL
LIN {X 0,Y 130.387,Z 866.684,A -85,B 0,C 180,E1 25823.838,E2 25823.838} C_VEL
LIN {X 0,Y 131.981,Z 866.072,A -85,B 0,C 180,E1 25829.713,E2 25829.713} C_VEL
LIN {X 0,Y 131.141,Z 864.577,A -85,B 0,C 180,E1 25833.935,E2 25833.935} C_VEL
LIN {X 0,Y 129.951,Z 860.557,A -85,B 0,C 180,E1 25841.091,E2 25841.091} C_VEL
LIN {X 0,Y 130.264,Z 854.701,A -85,B 0,C 180,E1 25848.344,E2 25848.344} C_VEL
LIN {X 0,Y 132.394,Z 846.894,A -85,B 0,C 180,E1 25855.498,E2 25855.498} C_VEL
LIN {X 0,Y 136.115,Z 837.589,A -85,B 0,C 180,E1 25861.931,E2 25861.931} C_VEL
LIN {X 0,Y 140.999,Z 826.841,A -85,B 0,C 180,E1 25867.579,E2 25867.579} C_VEL
LIN {X 0,Y 146.71,Z 814.631,A -85,B 0,C 180,E1 25872.432,E2 25872.432} C_VEL
LIN {X 0,Y 152.863,Z 800.807,A -85,B 0,C 180,E1 25876.556,E2 25876.556} C_VEL
LIN {X 0,Y 158.883,Z 785.997,A -85,B 0,C 180,E1 25879.873,E2 25879.873} C_VEL
LIN {X 0,Y 164.487,Z 770.265,A -85,B 0,C 180,E1 25882.493,E2 25882.493} C_VEL
LIN {X 0,Y 169.454,Z 753.394,A -85,B 0,C 180,E1 25884.516,E2 25884.516} C_VEL
LIN {X 0,Y 173.403,Z 735.726,A -85,B 0,C 180,E1 25886.011,E2 25886.011} C_VEL
LIN {X 0,Y 176.03,Z 717.762,A -85,B 0,C 180,E1 25887.045,E2 25887.045} C_VEL
LIN {X 0,Y 185.655,Z 590.84,A -85,B 0,C 180,E1 25891.14,E2 25891.14} C_VEL
LIN {X 0,Y 179.181,Z 576.95,A -85,B 0,C 180,E1 25894.377,E2 25894.377} C_VEL
LIN {X 0,Y 172.351,Z 564.092,A -85,B 0,C 180,E1 25898.206,E2 25898.206} C_VEL
LIN {X 0,Y 167.022,Z 555.438,A -85,B 0,C 180,E1 25901.593,E2 25901.593} C_VEL
LIN {X 0,Y 162.482,Z 548.64,A -85,B 0,C 180,E1 25904.84,E2 25904.84} C_VEL
LIN {X 0,Y 160.948,Z 546.008,A -85,B 0,C 180,E1 25906.346,E2 25906.346} C_VEL
LIN {X 0,Y 159.406,Z 541.519,A -85,B 0,C 180,E1 25910.615,E2 25910.615} C_VEL
LIN {X 0,Y 158.322,Z 538.388,A -85,B 0,C 180,E1 25914.201,E2 25914.201} C_VEL
LIN {X 0,Y 157.345,Z 535.57,A -85,B 0,C 180,E1 25918.18,E2 25918.18} C_VEL
LIN {X 0,Y 156.076,Z 532.098,A -85,B 0,C 180,E1 25925.515,E2 25925.515} C_VEL
LIN {X 0,Y 155.293,Z 531.101,A -85,B 0,C 180,E1 25932.268,E2 25932.268} C_VEL
LIN {X 0,Y 155.46,Z 531.444,A -85,B 0,C 180,E1 25939.149,E2 25939.149} C_VEL
LIN {X 0,Y 155.71,Z 532.412,A -85,B 0,C 180,E1 25942.662,E2 25942.662} C_VEL
LIN {X 0,Y 156.584,Z 535.321,A -85,B 0,C 180,E1 25949.033,E2 25949.033} C_VEL
LIN {X 0,Y 157.48,Z 538.767,A -85,B 0,C 180,E1 25953.969,E2 25953.969} C_VEL
LIN {X 0,Y 158.615,Z 542.848,A -85,B 0,C 180,E1 25958.615,E2 25958.615} C_VEL
LIN {X 0,Y 159.951,Z 548.19,A -85,B 0,C 180,E1 25963.52,E2 25963.52} C_VEL
LIN {X 0,Y 160.917,Z 550.496,A -85,B 0,C 180,E1 25964.85,E2 25964.85} C_VEL
LIN {X 0,Y 165.463,Z 558.146,A -85,B 0,C 180,E1 25968.297,E2 25968.297} C_VEL
LIN {X 0,Y 168.836,Z 564.22,A -85,B 0,C 180,E1 25970.61,E2 25970.61} C_VEL
LIN {X 0,Y 173.822,Z 574.074,A -85,B 0,C 180,E1 25973.711,E2 25973.711} C_VEL
LIN {X 0,Y 178.728,Z 585.298,A -85,B 0,C 180,E1 25976.506,E2 25976.506} C_VEL
LIN {X 0,Y 180.52,Z 616.987,A -85,B 0,C 180,E1 25979.144,E2 25979.144} C_VEL
LIN {X 0,Y 174.042,Z 698.087,A -85,B 0,C 180,E1 25981.965,E2 25981.965} C_VEL
LIN {X 0,Y 171.663,Z 715.542,A -85,B 0,C 180,E1 25983.13,E2 25983.13} C_VEL
LIN {X 0,Y 168.451,Z 731.395,A -85,B 0,C 180,E1 25984.699,E2 25984.699} C_VEL
LIN {X 0,Y 164.135,Z 747.251,A -85,B 0,C 180,E1 25986.906,E2 25986.906} C_VEL
LIN {X 0,Y 159.309,Z 761.712,A -85,B 0,C 180,E1 25989.606,E2 25989.606} C_VEL
LIN {X 0,Y 153.969,Z 775.287,A -85,B 0,C 180,E1 25993.008,E2 25993.008} C_VEL
LIN {X 0,Y 148.449,Z 787.795,A -85,B 0,C 180,E1 25997.157,E2 25997.157} C_VEL
LIN {X 0,Y 143.472,Z 798.2,A -85,B 0,C 180,E1 26001.738,E2 26001.738} C_VEL
LIN {X 0,Y 138.656,Z 808.016,A -85,B 0,C 180,E1 26007.519,E2 26007.519} C_VEL
LIN {X 0,Y 135.207,Z 815.4,A -85,B 0,C 180,E1 26013.391,E2 26013.391} C_VEL
LIN {X 0,Y 132.732,Z 821.703,A -85,B 0,C 180,E1 26020.415,E2 26020.415} C_VEL
LIN {X 0,Y 131.854,Z 826.116,A -85,B 0,C 180,E1 26027.656,E2 26027.656} C_VEL
LIN {X 0,Y 132.568,Z 828.65,A -85,B 0,C 180,E1 26034.983,E2 26034.983} C_VEL
LIN {X 0,Y 135.109,Z 829.46,A -85,B 0,C 180,E1 26042.471,E2 26042.471} C_VEL
LIN {X 0,Y 139.222,Z 828.445,A -85,B 0,C 180,E1 26049.196,E2 26049.196} C_VEL
LIN {X 0,Y 145.218,Z 825.535,A -85,B 0,C 180,E1 26055.729,E2 26055.729} C_VEL
LIN {X 0,Y 152.458,Z 820.906,A -85,B 0,C 180,E1 26061.461,E2 26061.461} C_VEL
LIN {X 0,Y 160.682,Z 814.433,A -85,B 0,C 180,E1 26066.493,E2 26066.493} C_VEL
LIN {X 0,Y 169.495,Z 806.291,A -85,B 0,C 180,E1 26070.815,E2 26070.815} C_VEL
LIN {X 0,Y 178.41,Z 796.576,A -85,B 0,C 180,E1 26074.46,E2 26074.46} C_VEL
LIN {X 0,Y 187.194,Z 785.307,A -85,B 0,C 180,E1 26077.523,E2 26077.523} C_VEL
LIN {X 0,Y 195.265,Z 773.087,A -85,B 0,C 180,E1 26079.985,E2 26079.985} C_VEL
LIN {X 0,Y 202.288,Z 760.239,A -85,B 0,C 180,E1 26081.935,E2 26081.935} C_VEL
LIN {X 0,Y 208.931,Z 745.212,A -85,B 0,C 180,E1 26083.653,E2 26083.653} C_VEL
LIN {X 0,Y 214.294,Z 729.63,A -85,B 0,C 180,E1 26084.977,E2 26084.977} C_VEL
LIN {X 0,Y 218.311,Z 713.185,A -85,B 0,C 180,E1 26085.977,E2 26085.977} C_VEL
LIN {X 0,Y 220.971,Z 695.85,A -85,B 0,C 180,E1 26086.685,E2 26086.685} C_VEL
LIN {X 0,Y 227.989,Z 628.678,A -85,B 0,C 180,E1 26088.425,E2 26088.425} C_VEL
LIN {X 0,Y 226.344,Z 623.732,A -85,B 0,C 180,E1 26090.336,E2 26090.336} C_VEL
LIN {X 0,Y 224.498,Z 618.757,A -85,B 0,C 180,E1 26092.836,E2 26092.836} C_VEL
LIN {X 0,Y 223.035,Z 614.982,A -85,B 0,C 180,E1 26095.242,E2 26095.242} C_VEL
LIN {X 0,Y 221.281,Z 610.234,A -85,B 0,C 180,E1 26099.482,E2 26099.482} C_VEL
LIN {X 0,Y 220.49,Z 607.682,A -85,B 0,C 180,E1 26105.203,E2 26105.203} C_VEL
LIN {X 0,Y 221.379,Z 608.428,A -85,B 0,C 180,E1 26110.145,E2 26110.145} C_VEL
LIN {X 0,Y 223.389,Z 611.934,A -85,B 0,C 180,E1 26114.648,E2 26114.648} C_VEL
LIN {X 0,Y 225.333,Z 615.548,A -85,B 0,C 180,E1 26117.561,E2 26117.561} C_VEL
LIN {X 0,Y 227.762,Z 620.365,A -85,B 0,C 180,E1 26120.426,E2 26120.426} C_VEL
LIN {X 0,Y 229.47,Z 624.115,A -85,B 0,C 180,E1 26122.161,E2 26122.161} C_VEL
LIN {X 0,Y 224.262,Z 675.367,A -85,B 0,C 180,E1 26123.38,E2 26123.38} C_VEL
LIN {X 0,Y 223.163,Z 683.054,A -85,B 0,C 180,E1 26123.319,E2 26123.319} C_VEL
LIN {X 0,Y 219.032,Z 703.511,A -85,B 0,C 180,E1 26122.281,E2 26122.281} C_VEL
LIN {X 0,Y 218.024,Z 710.091,A -85,B 0,C 180,E1 26122.271,E2 26122.271} C_VEL
LIN {X 0,Y 214.848,Z 728.039,A -85,B 0,C 180,E1 26122.841,E2 26122.841} C_VEL
LIN {X 0,Y 210.073,Z 745.133,A -85,B 0,C 180,E1 26123.621,E2 26123.621} C_VEL
LIN {X 0,Y 203.615,Z 762.138,A -85,B 0,C 180,E1 26124.709,E2 26124.709} C_VEL
LIN {X 0,Y 196.006,Z 777.987,A -85,B 0,C 180,E1 26126.13,E2 26126.13} C_VEL
LIN {X 0,Y 187.377,Z 792.737,A -85,B 0,C 180,E1 26127.98,E2 26127.98} C_VEL
LIN {X 0,Y 178.265,Z 805.937,A -85,B 0,C 180,E1 26130.26,E2 26130.26} C_VEL
LIN {X 0,Y 167.72,Z 819.165,A -85,B 0,C 180,E1 26133.426,E2 26133.426} C_VEL
LIN {X 0,Y 157.883,Z 830.045,A -85,B 0,C 180,E1 26137.067,E2 26137.067} C_VEL
LIN {X 0,Y 148.258,Z 839.608,A -85,B 0,C 180,E1 26141.533,E2 26141.533} C_VEL
LIN {X 0,Y 138.794,Z 848.243,A -85,B 0,C 180,E1 26147.378,E2 26147.378} C_VEL
LIN {X 0,Y 130.725,Z 855.29,A -85,B 0,C 180,E1 26154.459,E2 26154.459} C_VEL
LIN {X 0,Y 125.051,Z 860.42,A -85,B 0,C 180,E1 26162.372,E2 26162.372} C_VEL
LIN {X 0,Y 122.034,Z 863.735,A -85,B 0,C 180,E1 26170.87,E2 26170.87} C_VEL
LIN {X 0,Y 121.725,Z 865.279,A -85,B 0,C 180,E1 26179.59,E2 26179.59} C_VEL
LIN {X 0,Y 123.49,Z 865.096,A -85,B 0,C 180,E1 26187.681,E2 26187.681} C_VEL
LIN {X 0,Y 124.041,Z 864.585,A -85,B 0,C 180,E1 26190.463,E2 26190.463} C_VEL
LIN {X 0,Y 122.441,Z 861.58,A -85,B 0,C 180,E1 26197.508,E2 26197.508} C_VEL
LIN {X 0,Y 121.952,Z 856.611,A -85,B 0,C 180,E1 26205.211,E2 26205.211} C_VEL
LIN {X 0,Y 123.342,Z 849.762,A -85,B 0,C 180,E1 26212.9,E2 26212.9} C_VEL
LIN {X 0,Y 126.737,Z 840.856,A -85,B 0,C 180,E1 26220.326,E2 26220.326} C_VEL
LIN {X 0,Y 131.687,Z 830.341,A -85,B 0,C 180,E1 26226.858,E2 26226.858} C_VEL
LIN {X 0,Y 137.49,Z 818.586,A -85,B 0,C 180,E1 26232.276,E2 26232.276} C_VEL
LIN {X 0,Y 143.911,Z 805.286,A -85,B 0,C 180,E1 26236.847,E2 26236.847} C_VEL
LIN {X 0,Y 150.274,Z 790.987,A -85,B 0,C 180,E1 26240.518,E2 26240.518} C_VEL
LIN {X 0,Y 156.278,Z 775.765,A -85,B 0,C 180,E1 26243.413,E2 26243.413} C_VEL
LIN {X 0,Y 161.759,Z 759.167,A -85,B 0,C 180,E1 26245.698,E2 26245.698} C_VEL
LIN {X 0,Y 166.234,Z 742.17,A -85,B 0,C 180,E1 26247.36,E2 26247.36} C_VEL
LIN {X 0,Y 169.519,Z 724.31,A -85,B 0,C 180,E1 26248.584,E2 26248.584} C_VEL
LIN {X 0,Y 171.496,Z 705.264,A -85,B 0,C 180,E1 26249.381,E2 26249.381} C_VEL
LIN {X 0,Y 180.128,Z 593.566,A -85,B 0,C 180,E1 26252.969,E2 26252.969} C_VEL
LIN {X 0,Y 174.162,Z 580.638,A -85,B 0,C 180,E1 26256.216,E2 26256.216} C_VEL
LIN {X 0,Y 168.37,Z 569.443,A -85,B 0,C 180,E1 26259.766,E2 26259.766} C_VEL
LIN {X 0,Y 163.371,Z 561.059,A -85,B 0,C 180,E1 26263.192,E2 26263.192} C_VEL
LIN {X 0,Y 158.11,Z 552.89,A -85,B 0,C 180,E1 26267.399,E2 26267.399} C_VEL
LIN {X 0,Y 153.748,Z 546.624,A -85,B 0,C 180,E1 26271.775,E2 26271.775} C_VEL
LIN {X 0,Y 152.669,Z 543.559,A -85,B 0,C 180,E1 26275.493,E2 26275.493} C_VEL
LIN {X 0,Y 151.931,Z 541.328,A -85,B 0,C 180,E1 26278.869,E2 26278.869} C_VEL
LIN {X 0,Y 150.894,Z 538.18,A -85,B 0,C 180,E1 26285.705,E2 26285.705} C_VEL
LIN {X 0,Y 150.15,Z 537.23,A -85,B 0,C 180,E1 26292.304,E2 26292.304} C_VEL
LIN {X 0,Y 150.318,Z 537.594,A -85,B 0,C 180,E1 26299.426,E2 26299.426} C_VEL
LIN {X 0,Y 150.465,Z 538.537,A -85,B 0,C 180,E1 26302.671,E2 26302.671} C_VEL
LIN {X 0,Y 151.203,Z 541.293,A -85,B 0,C 180,E1 26308.864,E2 26308.864} C_VEL
LIN {X 0,Y 151.946,Z 544.444,A -85,B 0,C 180,E1 26313.557,E2 26313.557} C_VEL
LIN {X 0,Y 153.21,Z 548.943,A -85,B 0,C 180,E1 26318.674,E2 26318.674} C_VEL
LIN {X 0,Y 158.323,Z 557.457,A -85,B 0,C 180,E1 26323.752,E2 26323.752} C_VEL
LIN {X 0,Y 162.376,Z 564.626,A -85,B 0,C 180,E1 26327.055,E2 26327.055} C_VEL
LIN {X 0,Y 165.773,Z 571.033,A -85,B 0,C 180,E1 26329.529,E2 26329.529} C_VEL
LIN {X 0,Y 171.153,Z 582.331,A -85,B 0,C 180,E1 26333.086,E2 26333.086} C_VEL
LIN {X 0,Y 173.832,Z 589.247,A -85,B 0,C 180,E1 26334.764,E2 26334.764} C_VEL
LIN {X 0,Y 175.196,Z 618.034,A -85,B 0,C 180,E1 26337.228,E2 26337.228} C_VEL
LIN {X 0,Y 168.482,Z 698.758,A -85,B 0,C 180,E1 26340.049,E2 26340.049} C_VEL
LIN {X 0,Y 165.989,Z 716.223,A -85,B 0,C 180,E1 26341.227,E2 26341.227} C_VEL
LIN {X 0,Y 162.741,Z 731.622,A -85,B 0,C 180,E1 26342.759,E2 26342.759} C_VEL
LIN {X 0,Y 158.285,Z 747.421,A -85,B 0,C 180,E1 26344.961,E2 26344.961} C_VEL
LIN {X 0,Y 153.138,Z 762.202,A -85,B 0,C 180,E1 26347.747,E2 26347.747} C_VEL
LIN {X 0,Y 147.781,Z 775.278,A -85,B 0,C 180,E1 26351.048,E2 26351.048} C_VEL
LIN {X 0,Y 141.907,Z 787.94,A -85,B 0,C 180,E1 26355.306,E2 26355.306} C_VEL
LIN {X 0,Y 136.738,Z 798.251,A -85,B 0,C 180,E1 26359.892,E2 26359.892} C_VEL
LIN {X 0,Y 131.71,Z 807.881,A -85,B 0,C 180,E1 26365.645,E2 26365.645} C_VEL
LIN {X 0,Y 127.645,Z 816.007,A -85,B 0,C 180,E1 26372.244,E2 26372.244} C_VEL
LIN {X 0,Y 125.047,Z 822.133,A -85,B 0,C 180,E1 26379.201,E2 26379.201} C_VEL
LIN {X 0,Y 123.932,Z 826.767,A -85,B 0,C 180,E1 26386.883,E2 26386.883} C_VEL
LIN {X 0,Y 124.549,Z 829.61,A -85,B 0,C 180,E1 26394.673,E2 26394.673} C_VEL
LIN {X 0,Y 127.144,Z 830.643,A -85,B 0,C 180,E1 26402.705,E2 26402.705} C_VEL
LIN {X 0,Y 131.696,Z 829.822,A -85,B 0,C 180,E1 26410.19,E2 26410.19} C_VEL
LIN {X 0,Y 138.035,Z 827.066,A -85,B 0,C 180,E1 26417.019,E2 26417.019} C_VEL
LIN {X 0,Y 145.506,Z 822.701,A -85,B 0,C 180,E1 26422.853,E2 26422.853} C_VEL
LIN {X 0,Y 153.654,Z 816.904,A -85,B 0,C 180,E1 26427.771,E2 26427.771} C_VEL
LIN {X 0,Y 162.773,Z 809.137,A -85,B 0,C 180,E1 26432.194,E2 26432.194} C_VEL
LIN {X 0,Y 172.416,Z 799.458,A -85,B 0,C 180,E1 26436.049,E2 26436.049} C_VEL
LIN {X 0,Y 181.027,Z 789.288,A -85,B 0,C 180,E1 26438.975,E2 26438.975} C_VEL
LIN {X 0,Y 189.755,Z 777.006,A -85,B 0,C 180,E1 26441.569,E2 26441.569} C_VEL
LIN {X 0,Y 197.894,Z 763.215,A -85,B 0,C 180,E1 26443.733,E2 26443.733} C_VEL
LIN {X 0,Y 204.594,Z 749.177,A -85,B 0,C 180,E1 26445.381,E2 26445.381} C_VEL
LIN {X 0,Y 210.336,Z 733.771,A -85,B 0,C 180,E1 26446.73,E2 26446.73} C_VEL
LIN {X 0,Y 214.894,Z 717.22,A -85,B 0,C 180,E1 26447.788,E2 26447.788} C_VEL
LIN {X 0,Y 217.847,Z 700.565,A -85,B 0,C 180,E1 26448.514,E2 26448.514} C_VEL
LIN {X 0,Y 225.206,Z 632.938,A -85,B 0,C 180,E1 26450.244,E2 26450.244} C_VEL
LIN {X 0,Y 223.055,Z 626.492,A -85,B 0,C 180,E1 26453.307,E2 26453.307} C_VEL
LIN {X 0,Y 221.615,Z 622.49,A -85,B 0,C 180,E1 26455.86,E2 26455.86} C_VEL
LIN {X 0,Y 220.159,Z 618.133,A -85,B 0,C 180,E1 26459.739,E2 26459.739} C_VEL
LIN {X 0,Y 219.47,Z 615.616,A -85,B 0,C 180,E1 26465.227,E2 26465.227} C_VEL
LIN {X 0,Y 220.296,Z 616.343,A -85,B 0,C 180,E1 26469.972,E2 26469.972} C_VEL
LIN {X 0,Y 222.071,Z 619.647,A -85,B 0,C 180,E1 26474.204,E2 26474.204} C_VEL
LIN {X 0,Y 223.938,Z 623.357,A -85,B 0,C 180,E1 26477.161,E2 26477.161} C_VEL
LIN {X 0,Y 225.962,Z 627.654,A -85,B 0,C 180,E1 26479.718,E2 26479.718} C_VEL
LIN {X 0,Y 226.509,Z 629.158,A -85,B 0,C 180,E1 26480.359,E2 26480.359} C_VEL
LIN {X 0,Y 218.024,Z 710.091,A -85,B 0,C 180,E1 26482.271,E2 26482.271} C_VEL
LIN {X 0,Y 216.597,Z 717.731,A -85,B 0,C 180,E1 26482.239,E2 26482.239} C_VEL
LIN {X 0,Y 211.882,Z 732.453,A -85,B 0,C 180,E1 26481.54,E2 26481.54} C_VEL
LIN {X 0,Y 208.793,Z 740.79,A -85,B 0,C 180,E1 26481.394,E2 26481.394} C_VEL
LIN {X 0,Y 207.683,Z 743.908,A -85,B 0,C 180,E1 26481.497,E2 26481.497} C_VEL
LIN {X 0,Y 201.28,Z 760.525,A -85,B 0,C 180,E1 26482.49,E2 26482.49} C_VEL
LIN {X 0,Y 193.466,Z 776.513,A -85,B 0,C 180,E1 26483.83,E2 26483.83} C_VEL
LIN {X 0,Y 184.572,Z 791.391,A -85,B 0,C 180,E1 26485.585,E2 26485.585} C_VEL
LIN {X 0,Y 174.735,Z 805.162,A -85,B 0,C 180,E1 26487.864,E2 26487.864} C_VEL
LIN {X 0,Y 164.15,Z 817.892,A -85,B 0,C 180,E1 26490.813,E2 26490.813} C_VEL
LIN {X 0,Y 153.111,Z 829.487,A -85,B 0,C 180,E1 26494.634,E2 26494.634} C_VEL
LIN {X 0,Y 142.326,Z 839.444,A -85,B 0,C 180,E1 26499.398,E2 26499.398} C_VEL
LIN {X 0,Y 132.327,Z 847.874,A -85,B 0,C 180,E1 26505.357,E2 26505.357} C_VEL
LIN {X 0,Y 123.707,Z 854.728,A -85,B 0,C 180,E1 26512.687,E2 26512.687} C_VEL
LIN {X 0,Y 117.555,Z 859.614,A -85,B 0,C 180,E1 26521.001,E2 26521.001} C_VEL
LIN {X 0,Y 114.113,Z 862.819,A -85,B 0,C 180,E1 26530.553,E2 26530.553} C_VEL
LIN {X 0,Y 113.898,Z 864.124,A -85,B 0,C 180,E1 26540.4,E2 26540.4} C_VEL
LIN {X 0,Y 115.787,Z 863.639,A -85,B 0,C 180,E1 26548.516,E2 26548.516} C_VEL
LIN {X 0,Y 116.069,Z 863.223,A -85,B 0,C 180,E1 26550.494,E2 26550.494} C_VEL
LIN {X 0,Y 114.399,Z 860.092,A -85,B 0,C 180,E1 26558.04,E2 26558.04} C_VEL
LIN {X 0,Y 114.07,Z 854.971,A -85,B 0,C 180,E1 26566.29,E2 26566.29} C_VEL
LIN {X 0,Y 115.798,Z 847.972,A -85,B 0,C 180,E1 26574.486,E2 26574.486} C_VEL
LIN {X 0,Y 119.375,Z 839.519,A -85,B 0,C 180,E1 26581.85,E2 26581.85} C_VEL
LIN {X 0,Y 124.336,Z 829.701,A -85,B 0,C 180,E1 26588.259,E2 26588.259} C_VEL
LIN {X 0,Y 130.492,Z 818.022,A -85,B 0,C 180,E1 26593.926,E2 26593.926} C_VEL
LIN {X 0,Y 137.224,Z 804.822,A -85,B 0,C 180,E1 26598.634,E2 26598.634} C_VEL
LIN {X 0,Y 143.885,Z 790.591,A -85,B 0,C 180,E1 26602.392,E2 26602.392} C_VEL
LIN {X 0,Y 150.141,Z 775.474,A -85,B 0,C 180,E1 26605.332,E2 26605.332} C_VEL
LIN {X 0,Y 155.729,Z 759.352,A -85,B 0,C 180,E1 26607.598,E2 26607.598} C_VEL
LIN {X 0,Y 160.465,Z 742.184,A -85,B 0,C 180,E1 26609.304,E2 26609.304} C_VEL
LIN {X 0,Y 163.893,Z 724.483,A -85,B 0,C 180,E1 26610.539,E2 26610.539} C_VEL
LIN {X 0,Y 165.971,Z 706.053,A -85,B 0,C 180,E1 26611.341,E2 26611.341} C_VEL
LIN {X 0,Y 174.844,Z 596.539,A -85,B 0,C 180,E1 26614.859,E2 26614.859} C_VEL
LIN {X 0,Y 168.983,Z 583.571,A -85,B 0,C 180,E1 26618.388,E2 26618.388} C_VEL
LIN {X 0,Y 163.604,Z 573.203,A -85,B 0,C 180,E1 26622.024,E2 26622.024} C_VEL
LIN {X 0,Y 158.429,Z 564.359,A -85,B 0,C 180,E1 26626.032,E2 26626.032} C_VEL
LIN {X 0,Y 154.289,Z 557.971,A -85,B 0,C 180,E1 26629.82,E2 26629.82} C_VEL
LIN {X 0,Y 150.095,Z 551.926,A -85,B 0,C 180,E1 26634.458,E2 26634.458} C_VEL
LIN {X 0,Y 146.732,Z 547.297,A -85,B 0,C 180,E1 26639.415,E2 26639.415} C_VEL
LIN {X 0,Y 145.711,Z 544.261,A -85,B 0,C 180,E1 26645.909,E2 26645.909} C_VEL
LIN {X 0,Y 144.986,Z 543.349,A -85,B 0,C 180,E1 26652.75,E2 26652.75} C_VEL
LIN {X 0,Y 145.173,Z 543.74,A -85,B 0,C 180,E1 26659.724,E2 26659.724} C_VEL
LIN {X 0,Y 145.337,Z 545.527,A -85,B 0,C 180,E1 26664.814,E2 26664.814} C_VEL
LIN {X 0,Y 145.843,Z 547.279,A -85,B 0,C 180,E1 26668.68,E2 26668.68} C_VEL
LIN {X 0,Y 147.034,Z 549.966,A -85,B 0,C 180,E1 26672.149,E2 26672.149} C_VEL
LIN {X 0,Y 151.395,Z 556.827,A -85,B 0,C 180,E1 26678.015,E2 26678.015} C_VEL
LIN {X 0,Y 155.693,Z 564.24,A -85,B 0,C 180,E1 26682.526,E2 26682.526} C_VEL
LIN {X 0,Y 159.418,Z 571.208,A -85,B 0,C 180,E1 26685.811,E2 26685.811} C_VEL
LIN {X 0,Y 163.405,Z 579.116,A -85,B 0,C 180,E1 26688.886,E2 26688.886} C_VEL
LIN {X 0,Y 168.365,Z 590.663,A -85,B 0,C 180,E1 26692.381,E2 26692.381} C_VEL
LIN {X 0,Y 169.091,Z 593.058,A -85,B 0,C 180,E1 26692.904,E2 26692.904} C_VEL
LIN {X 0,Y 170.079,Z 618.96,A -85,B 0,C 180,E1 26695.194,E2 26695.194} C_VEL
LIN {X 0,Y 163.137,Z 699.15,A -85,B 0,C 180,E1 26697.996,E2 26697.996} C_VEL
LIN {X 0,Y 160.548,Z 716.604,A -85,B 0,C 180,E1 26699.173,E2 26699.173} C_VEL
LIN {X 0,Y 157.023,Z 732.598,A -85,B 0,C 180,E1 26700.775,E2 26700.775} C_VEL
LIN {X 0,Y 152.559,Z 747.747,A -85,B 0,C 180,E1 26702.902,E2 26702.902} C_VEL
LIN {X 0,Y 147.15,Z 762.622,A -85,B 0,C 180,E1 26705.726,E2 26705.726} C_VEL
LIN {X 0,Y 141.502,Z 775.812,A -85,B 0,C 180,E1 26709.093,E2 26709.093} C_VEL
LIN {X 0,Y 135.526,Z 788.066,A -85,B 0,C 180,E1 26713.277,E2 26713.277} C_VEL
LIN {X 0,Y 129.568,Z 799.325,A -85,B 0,C 180,E1 26718.425,E2 26718.425} C_VEL
LIN {X 0,Y 124.227,Z 808.954,A -85,B 0,C 180,E1 26724.457,E2 26724.457} C_VEL
LIN {X 0,Y 119.901,Z 817.088,A -85,B 0,C 180,E1 26731.433,E2 26731.433} C_VEL
LIN {X 0,Y 117.142,Z 823.233,A -85,B 0,C 180,E1 26738.837,E2 26738.837} C_VEL
LIN {X 0,Y 115.989,Z 827.892,A -85,B 0,C 180,E1 26747.042,E2 26747.042} C_VEL
LIN {X 0,Y 116.723,Z 830.771,A -85,B 0,C 180,E1 26755.359,E2 26755.359} C_VEL
LIN {X 0,Y 119.437,Z 831.831,A -85,B 0,C 180,E1 26763.539,E2 26763.539} C_VEL
LIN {X 0,Y 124.207,Z 831.146,A -85,B 0,C 180,E1 26771.306,E2 26771.306} C_VEL
LIN {X 0,Y 130.76,Z 828.687,A -85,B 0,C 180,E1 26778.298,E2 26778.298} C_VEL
LIN {X 0,Y 138.804,Z 824.412,A -85,B 0,C 180,E1 26784.486,E2 26784.486} C_VEL
LIN {X 0,Y 147.996,Z 818.359,A -85,B 0,C 180,E1 26789.855,E2 26789.855} C_VEL
LIN {X 0,Y 157.571,Z 810.718,A -85,B 0,C 180,E1 26794.296,E2 26794.296} C_VEL
LIN {X 0,Y 167.942,Z 800.837,A -85,B 0,C 180,E1 26798.241,E2 26798.241} C_VEL
LIN {X 0,Y 177.376,Z 790.165,A -85,B 0,C 180,E1 26801.262,E2 26801.262} C_VEL
LIN {X 0,Y 186.534,Z 777.71,A -85,B 0,C 180,E1 26803.815,E2 26803.815} C_VEL
LIN {X 0,Y 194.852,Z 764.055,A -85,B 0,C 180,E1 26805.888,E2 26805.888} C_VEL
LIN {X 0,Y 201.766,Z 750.002,A -85,B 0,C 180,E1 26807.483,E2 26807.483} C_VEL
LIN {X 0,Y 207.904,Z 733.963,A -85,B 0,C 180,E1 26808.835,E2 26808.835} C_VEL
LIN {X 0,Y 212.549,Z 717.483,A -85,B 0,C 180,E1 26809.845,E2 26809.845} C_VEL
LIN {X 0,Y 215.581,Z 700.593,A -85,B 0,C 180,E1 26810.55,E2 26810.55} C_VEL
LIN {X 0,Y 222.646,Z 637.627,A -85,B 0,C 180,E1 26812.127,E2 26812.127} C_VEL
LIN {X 0,Y 221.082,Z 632.628,A -85,B 0,C 180,E1 26814.745,E2 26814.745} C_VEL
LIN {X 0,Y 220.041,Z 629.545,A -85,B 0,C 180,E1 26816.874,E2 26816.874} C_VEL
LIN {X 0,Y 218.97,Z 625.794,A -85,B 0,C 180,E1 26820.297,E2 26820.297} C_VEL
LIN {X 0,Y 218.463,Z 623.545,A -85,B 0,C 180,E1 26825.515,E2 26825.515} C_VEL
LIN {X 0,Y 219.249,Z 624.338,A -85,B 0,C 180,E1 26829.924,E2 26829.924} C_VEL
LIN {X 0,Y 220.833,Z 627.511,A -85,B 0,C 180,E1 26833.884,E2 26833.884} C_VEL
LIN {X 0,Y 222.441,Z 630.898,A -85,B 0,C 180,E1 26836.584,E2 26836.584} C_VEL
LIN {X 0,Y 223.817,Z 634.021,A -85,B 0,C 180,E1 26838.506,E2 26838.506} C_VEL
LIN {X 0,Y 214.967,Z 714.106,A -85,B 0,C 180,E1 26840.364,E2 26840.364} C_VEL
LIN {X 0,Y 211.118,Z 732.32,A -85,B 0,C 180,E1 26840.976,E2 26840.976} C_VEL
LIN {X 0,Y 207.683,Z 743.908,A -85,B 0,C 180,E1 26841.497,E2 26841.497} C_VEL
LIN {X 0,Y 204.728,Z 751.269,A -85,B 0,C 180,E1 26841.634,E2 26841.634} C_VEL
LIN {X 0,Y 196.661,Z 765.905,A -85,B 0,C 180,E1 26841.228,E2 26841.228} C_VEL
LIN {X 0,Y 192.706,Z 772.503,A -85,B 0,C 180,E1 26841.304,E2 26841.304} C_VEL
LIN {X 0,Y 191.13,Z 775.26,A -85,B 0,C 180,E1 26841.495,E2 26841.495} C_VEL
LIN {X 0,Y 182.102,Z 790.042,A -85,B 0,C 180,E1 26843.121,E2 26843.121} C_VEL
LIN {X 0,Y 171.941,Z 803.87,A -85,B 0,C 180,E1 26845.279,E2 26845.279} C_VEL
LIN {X 0,Y 160.94,Z 816.64,A -85,B 0,C 180,E1 26848.094,E2 26848.094} C_VEL
LIN {X 0,Y 150.124,Z 827.537,A -85,B 0,C 180,E1 26851.515,E2 26851.515} C_VEL
LIN {X 0,Y 139.323,Z 837.111,A -85,B 0,C 180,E1 26855.812,E2 26855.812} C_VEL
LIN {X 0,Y 128.379,Z 845.739,A -85,B 0,C 180,E1 26861.612,E2 26861.612} C_VEL
LIN {X 0,Y 118.672,Z 852.795,A -85,B 0,C 180,E1 26868.916,E2 26868.916} C_VEL
LIN {X 0,Y 111.376,Z 857.916,A -85,B 0,C 180,E1 26877.41,E2 26877.41} C_VEL
LIN {X 0,Y 106.976,Z 861.203,A -85,B 0,C 180,E1 26886.887,E2 26886.887} C_VEL
LIN {X 0,Y 105.72,Z 862.772,A -85,B 0,C 180,E1 26897.437,E2 26897.437} C_VEL
LIN {X 0,Y 107.312,Z 862.523,A -85,B 0,C 180,E1 26906.796,E2 26906.796} C_VEL
LIN {X 0,Y 108.214,Z 862.026,A -85,B 0,C 180,E1 26910.001,E2 26910.001} C_VEL
LIN {X 0,Y 106.429,Z 858.869,A -85,B 0,C 180,E1 26918.102,E2 26918.102} C_VEL
LIN {X 0,Y 106.166,Z 853.716,A -85,B 0,C 180,E1 26926.976,E2 26926.976} C_VEL
LIN {X 0,Y 108.149,Z 846.673,A -85,B 0,C 180,E1 26935.756,E2 26935.756} C_VEL
LIN {X 0,Y 112.109,Z 838.159,A -85,B 0,C 180,E1 26943.571,E2 26943.571} C_VEL
LIN {X 0,Y 117.504,Z 828.26,A -85,B 0,C 180,E1 26950.294,E2 26950.294} C_VEL
LIN {X 0,Y 124.132,Z 816.441,A -85,B 0,C 180,E1 26956.156,E2 26956.156} C_VEL
LIN {X 0,Y 131.292,Z 803.122,A -85,B 0,C 180,E1 26960.969,E2 26960.969} C_VEL
LIN {X 0,Y 138.33,Z 788.741,A -85,B 0,C 180,E1 26964.764,E2 26964.764} C_VEL
LIN {X 0,Y 144.895,Z 773.319,A -85,B 0,C 180,E1 26967.708,E2 26967.708} C_VEL
LIN {X 0,Y 150.739,Z 756.83,A -85,B 0,C 180,E1 26969.954,E2 26969.954} C_VEL
LIN {X 0,Y 155.43,Z 740.002,A -85,B 0,C 180,E1 26971.574,E2 26971.574} C_VEL
LIN {X 0,Y 158.846,Z 722.397,A -85,B 0,C 180,E1 26972.762,E2 26972.762} C_VEL
LIN {X 0,Y 161.019,Z 702.396,A -85,B 0,C 180,E1 26973.579,E2 26973.579} C_VEL
LIN {X 0,Y 169.695,Z 599.455,A -85,B 0,C 180,E1 26976.899,E2 26976.899} C_VEL
LIN {X 0,Y 164.253,Z 587.121,A -85,B 0,C 180,E1 26980.533,E2 26980.533} C_VEL
LIN {X 0,Y 159.178,Z 577.106,A -85,B 0,C 180,E1 26984.331,E2 26984.331} C_VEL
LIN {X 0,Y 154.68,Z 569.281,A -85,B 0,C 180,E1 26988.252,E2 26988.252} C_VEL
LIN {X 0,Y 150.466,Z 562.576,A -85,B 0,C 180,E1 26992.651,E2 26992.651} C_VEL
LIN {X 0,Y 147.276,Z 558.116,A -85,B 0,C 180,E1 26996.712,E2 26996.712} C_VEL
LIN {X 0,Y 145.042,Z 554.763,A -85,B 0,C 180,E1 27000.396,E2 27000.396} C_VEL
LIN {X 0,Y 142.406,Z 551.479,A -85,B 0,C 180,E1 27006.451,E2 27006.451} C_VEL
LIN {X 0,Y 141.056,Z 550.319,A -85,B 0,C 180,E1 27013.111,E2 27013.111} C_VEL
LIN {X 0,Y 141.314,Z 550.769,A -85,B 0,C 180,E1 27019.855,E2 27019.855} C_VEL
LIN {X 0,Y 143.863,Z 554.97,A -85,B 0,C 180,E1 27028.205,E2 27028.205} C_VEL
LIN {X 0,Y 145.879,Z 558.459,A -85,B 0,C 180,E1 27032.087,E2 27032.087} C_VEL
LIN {X 0,Y 149.236,Z 563.91,A -85,B 0,C 180,E1 27036.845,E2 27036.845} C_VEL
LIN {X 0,Y 153.045,Z 570.842,A -85,B 0,C 180,E1 27041.165,E2 27041.165} C_VEL
LIN {X 0,Y 156.684,Z 578.068,A -85,B 0,C 180,E1 27044.649,E2 27044.649} C_VEL
LIN {X 0,Y 160.62,Z 586.612,A -85,B 0,C 180,E1 27047.932,E2 27047.932} C_VEL
LIN {X 0,Y 164.517,Z 596.283,A -85,B 0,C 180,E1 27050.882,E2 27050.882} C_VEL
LIN {X 0,Y 165.176,Z 620.024,A -85,B 0,C 180,E1 27053.041,E2 27053.041} C_VEL
LIN {X 0,Y 157.997,Z 699.698,A -85,B 0,C 180,E1 27055.816,E2 27055.816} C_VEL
LIN {X 0,Y 155.285,Z 717.195,A -85,B 0,C 180,E1 27056.996,E2 27056.996} C_VEL
LIN {X 0,Y 151.607,Z 733.192,A -85,B 0,C 180,E1 27058.599,E2 27058.599} C_VEL
LIN {X 0,Y 146.721,Z 748.989,A -85,B 0,C 180,E1 27060.839,E2 27060.839} C_VEL
LIN {X 0,Y 141.053,Z 763.795,A -85,B 0,C 180,E1 27063.702,E2 27063.702} C_VEL
LIN {X 0,Y 135.114,Z 776.921,A -85,B 0,C 180,E1 27067.138,E2 27067.138} C_VEL
LIN {X 0,Y 128.505,Z 789.715,A -85,B 0,C 180,E1 27071.67,E2 27071.67} C_VEL
LIN {X 0,Y 122.491,Z 800.4,A -85,B 0,C 180,E1 27076.787,E2 27076.787} C_VEL
LIN {X 0,Y 116.804,Z 810.026,A -85,B 0,C 180,E1 27083.116,E2 27083.116} C_VEL
LIN {X 0,Y 112.185,Z 818.169,A -85,B 0,C 180,E1 27090.51,E2 27090.51} C_VEL
LIN {X 0,Y 109.205,Z 824.424,A -85,B 0,C 180,E1 27098.565,E2 27098.565} C_VEL
LIN {X 0,Y 108.042,Z 829.174,A -85,B 0,C 180,E1 27107.594,E2 27107.594} C_VEL
LIN {X 0,Y 108.915,Z 831.929,A -85,B 0,C 180,E1 27116.144,E2 27116.144} C_VEL
LIN {X 0,Y 111.939,Z 833.027,A -85,B 0,C 180,E1 27124.865,E2 27124.865} C_VEL
LIN {X 0,Y 117.162,Z 832.385,A -85,B 0,C 180,E1 27133.055,E2 27133.055} C_VEL
LIN {X 0,Y 124.422,Z 829.917,A -85,B 0,C 180,E1 27140.484,E2 27140.484} C_VEL
LIN {X 0,Y 133.439,Z 825.45,A -85,B 0,C 180,E1 27147.056,E2 27147.056} C_VEL
LIN {X 0,Y 143.239,Z 819.356,A -85,B 0,C 180,E1 27152.436,E2 27152.436} C_VEL
LIN {X 0,Y 153.342,Z 811.661,A -85,B 0,C 180,E1 27156.834,E2 27156.834} C_VEL
LIN {X 0,Y 164.203,Z 801.751,A -85,B 0,C 180,E1 27160.702,E2 27160.702} C_VEL
LIN {X 0,Y 174.055,Z 790.996,A -85,B 0,C 180,E1 27163.651,E2 27163.651} C_VEL
LIN {X 0,Y 183.624,Z 778.423,A -85,B 0,C 180,E1 27166.137,E2 27166.137} C_VEL
LIN {X 0,Y 192.097,Z 764.965,A -85,B 0,C 180,E1 27168.105,E2 27168.105} C_VEL
LIN {X 0,Y 199.221,Z 750.968,A -85,B 0,C 180,E1 27169.636,E2 27169.636} C_VEL
LIN {X 0,Y 205.311,Z 735.658,A -85,B 0,C 180,E1 27170.888,E2 27170.888} C_VEL
LIN {X 0,Y 210.2,Z 719.057,A -85,B 0,C 180,E1 27171.883,E2 27171.883} C_VEL
LIN {X 0,Y 213.4,Z 702.424,A -85,B 0,C 180,E1 27172.571,E2 27172.571} C_VEL
LIN {X 0,Y 220.351,Z 642.524,A -85,B 0,C 180,E1 27174.009,E2 27174.009} C_VEL
LIN {X 0,Y 218.912,Z 637.652,A -85,B 0,C 180,E1 27176.989,E2 27176.989} C_VEL
LIN {X 0,Y 217.813,Z 633.541,A -85,B 0,C 180,E1 27180.789,E2 27180.789} C_VEL
LIN {X 0,Y 217.444,Z 631.48,A -85,B 0,C 180,E1 27185.541,E2 27185.541} C_VEL
LIN {X 0,Y 218.172,Z 632.264,A -85,B 0,C 180,E1 27189.762,E2 27189.762} C_VEL
LIN {X 0,Y 219.601,Z 635.372,A -85,B 0,C 180,E1 27193.561,E2 27193.561} C_VEL
LIN {X 0,Y 221.061,Z 638.662,A -85,B 0,C 180,E1 27196.15,E2 27196.15} C_VEL
LIN {X 0,Y 221.341,Z 639.538,A -85,B 0,C 180,E1 27196.62,E2 27196.62} C_VEL
LIN {X 0,Y 212.901,Z 713.342,A -85,B 0,C 180,E1 27198.279,E2 27198.279} C_VEL
LIN {X 0,Y 208.995,Z 731.402,A -85,B 0,C 180,E1 27198.853,E2 27198.853} C_VEL
LIN {X 0,Y 203.475,Z 748.669,A -85,B 0,C 180,E1 27199.623,E2 27199.623} C_VEL
LIN {X 0,Y 196.576,Z 764.755,A -85,B 0,C 180,E1 27200.628,E2 27200.628} C_VEL
LIN {X 0,Y 191.13,Z 775.26,A -85,B 0,C 180,E1 27201.495,E2 27201.495} C_VEL
LIN {X 0,Y 187.038,Z 781.763,A -85,B 0,C 180,E1 27201.853,E2 27201.853} C_VEL
LIN {X 0,Y 176.397,Z 794.731,A -85,B 0,C 180,E1 27201.951,E2 27201.951} C_VEL
LIN {X 0,Y 171.301,Z 800.499,A -85,B 0,C 180,E1 27202.325,E2 27202.325} C_VEL
LIN {X 0,Y 169.249,Z 802.891,A -85,B 0,C 180,E1 27202.671,E2 27202.671} C_VEL
LIN {X 0,Y 158.111,Z 815.385,A -85,B 0,C 180,E1 27205.272,E2 27205.272} C_VEL
LIN {X 0,Y 146.817,Z 826.307,A -85,B 0,C 180,E1 27208.537,E2 27208.537} C_VEL
LIN {X 0,Y 135.435,Z 835.894,A -85,B 0,C 180,E1 27212.69,E2 27212.69} C_VEL
LIN {X 0,Y 123.726,Z 844.523,A -85,B 0,C 180,E1 27218.384,E2 27218.384} C_VEL
LIN {X 0,Y 113.132,Z 851.553,A -85,B 0,C 180,E1 27225.718,E2 27225.718} C_VEL
LIN {X 0,Y 104.915,Z 856.666,A -85,B 0,C 180,E1 27234.456,E2 27234.456} C_VEL
LIN {X 0,Y 99.631,Z 859.965,A -85,B 0,C 180,E1 27244.58,E2 27244.58} C_VEL
LIN {X 0,Y 97.767,Z 861.501,A -85,B 0,C 180,E1 27255.793,E2 27255.793} C_VEL
LIN {X 0,Y 99.279,Z 861.194,A -85,B 0,C 180,E1 27266.537,E2 27266.537} C_VEL
LIN {X 0,Y 100.216,Z 860.653,A -85,B 0,C 180,E1 27270.001,E2 27270.001} C_VEL
LIN {X 0,Y 98.381,Z 857.351,A -85,B 0,C 180,E1 27278.77,E2 27278.77} C_VEL
LIN {X 0,Y 98.432,Z 851.66,A -85,B 0,C 180,E1 27288.97,E2 27288.97} C_VEL
LIN {X 0,Y 101.023,Z 844.342,A -85,B 0,C 180,E1 27298.365,E2 27298.365} C_VEL
LIN {X 0,Y 105.701,Z 835.474,A -85,B 0,C 180,E1 27306.581,E2 27306.581} C_VEL
LIN {X 0,Y 111.975,Z 824.863,A -85,B 0,C 180,E1 27313.676,E2 27313.676} C_VEL
LIN {X 0,Y 119.413,Z 812.434,A -85,B 0,C 180,E1 27319.638,E2 27319.638} C_VEL
LIN {X 0,Y 126.903,Z 799.022,A -85,B 0,C 180,E1 27324.247,E2 27324.247} C_VEL
LIN {X 0,Y 134.093,Z 784.564,A -85,B 0,C 180,E1 27327.814,E2 27327.814} C_VEL
LIN {X 0,Y 140.669,Z 769.254,A -85,B 0,C 180,E1 27330.543,E2 27330.543} C_VEL
LIN {X 0,Y 146.626,Z 752.472,A -85,B 0,C 180,E1 27332.671,E2 27332.671} C_VEL
LIN {X 0,Y 151.233,Z 735.22,A -85,B 0,C 180,E1 27334.183,E2 27334.183} C_VEL
LIN {X 0,Y 154.507,Z 716.764,A -85,B 0,C 180,E1 27335.288,E2 27335.288} C_VEL
LIN {X 0,Y 158.297,Z 675.912,A -85,B 0,C 180,E1 27336.7,E2 27336.7} C_VEL
LIN {X 0,Y 164.815,Z 602.536,A -85,B 0,C 180,E1 27339.028,E2 27339.028} C_VEL
LIN {X 0,Y 159.798,Z 590.978,A -85,B 0,C 180,E1 27342.711,E2 27342.711} C_VEL
LIN {X 0,Y 154.989,Z 581.297,A -85,B 0,C 180,E1 27346.762,E2 27346.762} C_VEL
LIN {X 0,Y 150.572,Z 573.26,A -85,B 0,C 180,E1 27351.216,E2 27351.216} C_VEL
LIN {X 0,Y 146.485,Z 566.793,A -85,B 0,C 180,E1 27356.283,E2 27356.283} C_VEL
LIN {X 0,Y 143.568,Z 562.373,A -85,B 0,C 180,E1 27361.198,E2 27361.198} C_VEL
LIN {X 0,Y 141.243,Z 559.318,A -85,B 0,C 180,E1 27366.913,E2 27366.913} C_VEL
LIN {X 0,Y 140.016,Z 558.229,A -85,B 0,C 180,E1 27373.786,E2 27373.786} C_VEL
LIN {X 0,Y 140.334,Z 558.77,A -85,B 0,C 180,E1 27379.999,E2 27379.999} C_VEL
LIN {X 0,Y 142.628,Z 562.874,A -85,B 0,C 180,E1 27387.788,E2 27387.788} C_VEL
LIN {X 0,Y 144.441,Z 566.322,A -85,B 0,C 180,E1 27391.51,E2 27391.51} C_VEL
LIN {X 0,Y 147.212,Z 571.145,A -85,B 0,C 180,E1 27395.741,E2 27395.741} C_VEL
LIN {X 0,Y 150.57,Z 577.638,A -85,B 0,C 180,E1 27399.853,E2 27399.853} C_VEL
LIN {X 0,Y 154.295,Z 585.482,A -85,B 0,C 180,E1 27403.707,E2 27403.707} C_VEL
LIN {X 0,Y 158.593,Z 595.792,A -85,B 0,C 180,E1 27407.531,E2 27407.531} C_VEL
LIN {X 0,Y 160.146,Z 600.445,A -85,B 0,C 180,E1 27408.845,E2 27408.845} C_VEL
LIN {X 0,Y 160.528,Z 621.003,A -85,B 0,C 180,E1 27410.758,E2 27410.758} C_VEL
LIN {X 0,Y 153.078,Z 700.408,A -85,B 0,C 180,E1 27413.501,E2 27413.501} C_VEL
LIN {X 0,Y 150.242,Z 717.888,A -85,B 0,C 180,E1 27414.679,E2 27414.679} C_VEL
LIN {X 0,Y 146.202,Z 734.585,A -85,B 0,C 180,E1 27416.361,E2 27416.361} C_VEL
LIN {X 0,Y 141.09,Z 750.231,A -85,B 0,C 180,E1 27418.608,E2 27418.608} C_VEL
LIN {X 0,Y 135.149,Z 764.967,A -85,B 0,C 180,E1 27421.498,E2 27421.498} C_VEL
LIN {X 0,Y 128.597,Z 778.604,A -85,B 0,C 180,E1 27425.174,E2 27425.174} C_VEL
LIN {X 0,Y 121.688,Z 791.203,A -85,B 0,C 180,E1 27429.811,E2 27429.811} C_VEL
LIN {X 0,Y 115.049,Z 802.219,A -85,B 0,C 180,E1 27435.401,E2 27435.401} C_VEL
LIN {X 0,Y 108.997,Z 811.824,A -85,B 0,C 180,E1 27442.194,E2 27442.194} C_VEL
LIN {X 0,Y 104.232,Z 819.728,A -85,B 0,C 180,E1 27449.999,E2 27449.999} C_VEL
LIN {X 0,Y 101.069,Z 826.1,A -85,B 0,C 180,E1 27459.106,E2 27459.106} C_VEL
LIN {X 0,Y 100.108,Z 830.611,A -85,B 0,C 180,E1 27468.638,E2 27468.638} C_VEL
LIN {X 0,Y 101.419,Z 833.297,A -85,B 0,C 180,E1 27478.242,E2 27478.242} C_VEL
LIN {X 0,Y 105.412,Z 834.251,A -85,B 0,C 180,E1 27488.066,E2 27488.066} C_VEL
LIN {X 0,Y 111.56,Z 833.333,A -85,B 0,C 180,E1 27496.548,E2 27496.548} C_VEL
LIN {X 0,Y 119.765,Z 830.53,A -85,B 0,C 180,E1 27504.076,E2 27504.076} C_VEL
LIN {X 0,Y 129.693,Z 825.806,A -85,B 0,C 180,E1 27510.593,E2 27510.593} C_VEL
LIN {X 0,Y 140.261,Z 819.335,A -85,B 0,C 180,E1 27515.845,E2 27515.845} C_VEL
LIN {X 0,Y 151.015,Z 811.338,A -85,B 0,C 180,E1 27520.078,E2 27520.078} C_VEL
LIN {X 0,Y 161.618,Z 801.914,A -85,B 0,C 180,E1 27523.518,E2 27523.518} C_VEL
LIN {X 0,Y 171.845,Z 790.957,A -85,B 0,C 180,E1 27526.327,E2 27526.327} C_VEL
LIN {X 0,Y 181.978,Z 777.888,A -85,B 0,C 180,E1 27528.737,E2 27528.737} C_VEL
LIN {X 0,Y 190.55,Z 764.357,A -85,B 0,C 180,E1 27530.565,E2 27530.565} C_VEL
LIN {X 0,Y 197.887,Z 749.892,A -85,B 0,C 180,E1 27532.021,E2 27532.021} C_VEL
LIN {X 0,Y 204.153,Z 734.058,A -85,B 0,C 180,E1 27533.208,E2 27533.208} C_VEL
LIN {X 0,Y 208.827,Z 717.815,A -85,B 0,C 180,E1 27534.097,E2 27534.097} C_VEL
LIN {X 0,Y 211.974,Z 700.653,A -85,B 0,C 180,E1 27534.744,E2 27534.744} C_VEL
LIN {X 0,Y 218.223,Z 647.687,A -85,B 0,C 180,E1 27535.986,E2 27535.986} C_VEL
LIN {X 0,Y 217.396,Z 644.559,A -85,B 0,C 180,E1 27538.155,E2 27538.155} C_VEL
LIN {X 0,Y 216.719,Z 641.402,A -85,B 0,C 180,E1 27541.057,E2 27541.057} C_VEL
LIN {X 0,Y 216.425,Z 639.415,A -85,B 0,C 180,E1 27545.567,E2 27545.567} C_VEL
LIN {X 0,Y 217.083,Z 640.156,A -85,B 0,C 180,E1 27549.544,E2 27549.544} C_VEL
LIN {X 0,Y 218.319,Z 643.081,A -85,B 0,C 180,E1 27553.102,E2 27553.102} C_VEL
LIN {X 0,Y 219.106,Z 645.084,A -85,B 0,C 180,E1 27554.695,E2 27554.695} C_VEL
LIN {X 0,Y 211.124,Z 712.78,A -85,B 0,C 180,E1 27556.159,E2 27556.159} C_VEL
LIN {X 0,Y 207.083,Z 730.99,A -85,B 0,C 180,E1 27556.703,E2 27556.703} C_VEL
LIN {X 0,Y 201.687,Z 747.528,A -85,B 0,C 180,E1 27557.387,E2 27557.387} C_VEL
LIN {X 0,Y 194.816,Z 763.338,A -85,B 0,C 180,E1 27558.291,E2 27558.291} C_VEL
LIN {X 0,Y 186.219,Z 779.016,A -85,B 0,C 180,E1 27559.559,E2 27559.559} C_VEL
LIN {X 0,Y 176.417,Z 793.687,A -85,B 0,C 180,E1 27561.248,E2 27561.248} C_VEL
LIN {X 0,Y 169.249,Z 802.891,A -85,B 0,C 180,E1 27562.671,E2 27562.671} C_VEL
LIN {X 0,Y 164.101,Z 808.422,A -85,B 0,C 180,E1 27563.394,E2 27563.394} C_VEL
LIN {X 0,Y 152.261,Z 818.482,A -85,B 0,C 180,E1 27564.178,E2 27564.178} C_VEL
LIN {X 0,Y 145.555,Z 823.734,A -85,B 0,C 180,E1 27565.061,E2 27565.061} C_VEL
LIN {X 0,Y 143.283,Z 825.647,A -85,B 0,C 180,E1 27565.622,E2 27565.622} C_VEL
LIN {X 0,Y 131.191,Z 835.244,A -85,B 0,C 180,E1 27569.695,E2 27569.695} C_VEL
LIN {X 0,Y 118.808,Z 843.747,A -85,B 0,C 180,E1 27575.283,E2 27575.283} C_VEL
LIN {X 0,Y 107.404,Z 850.675,A -85,B 0,C 180,E1 27582.657,E2 27582.657} C_VEL
LIN {X 0,Y 98.341,Z 855.645,A -85,B 0,C 180,E1 27591.67,E2 27591.67} C_VEL
LIN {X 0,Y 92.096,Z 858.916,A -85,B 0,C 180,E1 27602.902,E2 27602.902} C_VEL
LIN {X 0,Y 89.861,Z 860.289,A -85,B 0,C 180,E1 27615.173,E2 27615.173} C_VEL
LIN {X 0,Y 91.399,Z 859.798,A -85,B 0,C 180,E1 27626.866,E2 27626.866} C_VEL
LIN {X 0,Y 92.198,Z 859.269,A -85,B 0,C 180,E1 27630.001,E2 27630.001} C_VEL
LIN {X 0,Y 90.311,Z 855.707,A -85,B 0,C 180,E1 27639.826,E2 27639.826} C_VEL
LIN {X 0,Y 90.702,Z 849.986,A -85,B 0,C 180,E1 27650.657,E2 27650.657} C_VEL
LIN {X 0,Y 93.848,Z 842.465,A -85,B 0,C 180,E1 27660.758,E2 27660.758} C_VEL
LIN {X 0,Y 99.188,Z 833.374,A -85,B 0,C 180,E1 27669.427,E2 27669.427} C_VEL
LIN {X 0,Y 105.962,Z 822.825,A -85,B 0,C 180,E1 27676.601,E2 27676.601} C_VEL
LIN {X 0,Y 113.779,Z 810.572,A -85,B 0,C 180,E1 27682.505,E2 27682.505} C_VEL
LIN {X 0,Y 121.559,Z 797.251,A -85,B 0,C 180,E1 27687.034,E2 27687.034} C_VEL
LIN {X 0,Y 129.137,Z 782.619,A -85,B 0,C 180,E1 27690.582,E2 27690.582} C_VEL
LIN {X 0,Y 136.128,Z 766.83,A -85,B 0,C 180,E1 27693.302,E2 27693.302} C_VEL
LIN {X 0,Y 142.002,Z 750.467,A -85,B 0,C 180,E1 27695.274,E2 27695.274} C_VEL
LIN {X 0,Y 146.674,Z 733.103,A -85,B 0,C 180,E1 27696.73,E2 27696.73} C_VEL
LIN {X 0,Y 149.883,Z 715.128,A -85,B 0,C 180,E1 27697.76,E2 27697.76} C_VEL
LIN {X 0,Y 160.104,Z 605.668,A -85,B 0,C 180,E1 27701.287,E2 27701.287} C_VEL
LIN {X 0,Y 155.199,Z 593.992,A -85,B 0,C 180,E1 27705.354,E2 27705.354} C_VEL
LIN {X 0,Y 150.837,Z 585.006,A -85,B 0,C 180,E1 27709.594,E2 27709.594} C_VEL
LIN {X 0,Y 147.5,Z 579,A -85,B 0,C 180,E1 27713.383,E2 27713.383} C_VEL
LIN {X 0,Y 144.608,Z 574.055,A -85,B 0,C 180,E1 27717.425,E2 27717.425} C_VEL
LIN {X 0,Y 142.078,Z 569.931,A -85,B 0,C 180,E1 27722.108,E2 27722.108} C_VEL
LIN {X 0,Y 140.09,Z 567.158,A -85,B 0,C 180,E1 27727.382,E2 27727.382} C_VEL
LIN {X 0,Y 139.003,Z 566.154,A -85,B 0,C 180,E1 27734.157,E2 27734.157} C_VEL
LIN {X 0,Y 139.308,Z 566.771,A -85,B 0,C 180,E1 27739.907,E2 27739.907} C_VEL
LIN {X 0,Y 141.316,Z 570.622,A -85,B 0,C 180,E1 27747.153,E2 27747.153} C_VEL
LIN {X 0,Y 143.777,Z 575.478,A -85,B 0,C 180,E1 27752.259,E2 27752.259} C_VEL
LIN {X 0,Y 145.781,Z 579.509,A -85,B 0,C 180,E1 27755.396,E2 27755.396} C_VEL
LIN {X 0,Y 148.237,Z 584.621,A -85,B 0,C 180,E1 27758.603,E2 27758.603} C_VEL
LIN {X 0,Y 151.651,Z 592.273,A -85,B 0,C 180,E1 27762.436,E2 27762.436} C_VEL
LIN {X 0,Y 155.952,Z 603.651,A -85,B 0,C 180,E1 27766.607,E2 27766.607} C_VEL
LIN {X 0,Y 156.089,Z 622.008,A -85,B 0,C 180,E1 27768.356,E2 27768.356} C_VEL
LIN {X 0,Y 148.396,Z 700.991,A -85,B 0,C 180,E1 27771.043,E2 27771.043} C_VEL
LIN {X 0,Y 145.44,Z 718.468,A -85,B 0,C 180,E1 27772.207,E2 27772.207} C_VEL
LIN {X 0,Y 141.39,Z 734.626,A -85,B 0,C 180,E1 27773.808,E2 27773.808} C_VEL
LIN {X 0,Y 136.038,Z 750.459,A -85,B 0,C 180,E1 27776.041,E2 27776.041} C_VEL
LIN {X 0,Y 129.796,Z 765.304,A -85,B 0,C 180,E1 27778.926,E2 27778.926} C_VEL
LIN {X 0,Y 123.201,Z 778.499,A -85,B 0,C 180,E1 27782.444,E2 27782.444} C_VEL
LIN {X 0,Y 115.831,Z 791.268,A -85,B 0,C 180,E1 27787.141,E2 27787.141} C_VEL
LIN {X 0,Y 108.691,Z 802.497,A -85,B 0,C 180,E1 27792.879,E2 27792.879} C_VEL
LIN {X 0,Y 102.187,Z 812.128,A -85,B 0,C 180,E1 27799.855,E2 27799.855} C_VEL
LIN {X 0,Y 96.852,Z 820.29,A -85,B 0,C 180,E1 27808.224,E2 27808.224} C_VEL
LIN {X 0,Y 93.46,Z 826.502,A -85,B 0,C 180,E1 27817.375,E2 27817.375} C_VEL
LIN {X 0,Y 92.161,Z 831.236,A -85,B 0,C 180,E1 27827.683,E2 27827.683} C_VEL
LIN {X 0,Y 93.372,Z 834.22,A -85,B 0,C 180,E1 27838.109,E2 27838.109} C_VEL
LIN {X 0,Y 97.165,Z 835.419,A -85,B 0,C 180,E1 27848.127,E2 27848.127} C_VEL
LIN {X 0,Y 103.936,Z 834.779,A -85,B 0,C 180,E1 27857.793,E2 27857.793} C_VEL
LIN {X 0,Y 112.551,Z 832.31,A -85,B 0,C 180,E1 27865.706,E2 27865.706} C_VEL
LIN {X 0,Y 122.923,Z 827.865,A -85,B 0,C 180,E1 27872.448,E2 27872.448} C_VEL
LIN {X 0,Y 133.92,Z 821.826,A -85,B 0,C 180,E1 27877.787,E2 27877.787} C_VEL
LIN {X 0,Y 145.049,Z 814.238,A -85,B 0,C 180,E1 27882.037,E2 27882.037} C_VEL
LIN {X 0,Y 156.836,Z 804.451,A -85,B 0,C 180,E1 27885.7,E2 27885.7} C_VEL
LIN {X 0,Y 167.82,Z 793.454,A -85,B 0,C 180,E1 27888.541,E2 27888.541} C_VEL
LIN {X 0,Y 177.775,Z 781.327,A -85,B 0,C 180,E1 27890.771,E2 27890.771} C_VEL
LIN {X 0,Y 187.06,Z 767.573,A -85,B 0,C 180,E1 27892.629,E2 27892.629} C_VEL
LIN {X 0,Y 195.007,Z 752.945,A -85,B 0,C 180,E1 27894.091,E2 27894.091} C_VEL
LIN {X 0,Y 201.658,Z 737.071,A -85,B 0,C 180,E1 27895.264,E2 27895.264} C_VEL
LIN {X 0,Y 206.795,Z 720.464,A -85,B 0,C 180,E1 27896.164,E2 27896.164} C_VEL
LIN {X 0,Y 210.195,Z 703.665,A -85,B 0,C 180,E1 27896.799,E2 27896.799} C_VEL
LIN {X 0,Y 216.39,Z 653.049,A -85,B 0,C 180,E1 27897.941,E2 27897.941} C_VEL
LIN {X 0,Y 215.58,Z 649.13,A -85,B 0,C 180,E1 27901.594,E2 27901.594} C_VEL
LIN {X 0,Y 215.425,Z 647.355,A -85,B 0,C 180,E1 27905.86,E2 27905.86} C_VEL
LIN {X 0,Y 215.998,Z 648.047,A -85,B 0,C 180,E1 27909.323,E2 27909.323} C_VEL
LIN {X 0,Y 217.092,Z 650.899,A -85,B 0,C 180,E1 27912.737,E2 27912.737} C_VEL
LIN {X 0,Y 209.656,Z 712.131,A -85,B 0,C 180,E1 27914.004,E2 27914.004} C_VEL
LIN {X 0,Y 205.525,Z 730.364,A -85,B 0,C 180,E1 27914.509,E2 27914.509} C_VEL
LIN {X 0,Y 199.918,Z 747.174,A -85,B 0,C 180,E1 27915.149,E2 27915.149} C_VEL
LIN {X 0,Y 192.458,Z 763.744,A -85,B 0,C 180,E1 27916.032,E2 27916.032} C_VEL
LIN {X 0,Y 183.869,Z 778.902,A -85,B 0,C 180,E1 27917.178,E2 27917.178} C_VEL
LIN {X 0,Y 174.158,Z 792.995,A -85,B 0,C 180,E1 27918.689,E2 27918.689} C_VEL
LIN {X 0,Y 163.495,Z 805.952,A -85,B 0,C 180,E1 27920.664,E2 27920.664} C_VEL
LIN {X 0,Y 151.424,Z 818.296,A -85,B 0,C 180,E1 27923.392,E2 27923.392} C_VEL
LIN {X 0,Y 143.283,Z 825.647,A -85,B 0,C 180,E1 27925.622,E2 27925.622} C_VEL
LIN {X 0,Y 137.603,Z 829.959,A -85,B 0,C 180,E1 27926.879,E2 27926.879} C_VEL
LIN {X 0,Y 122.693,Z 838.37,A -85,B 0,C 180,E1 27929.19,E2 27929.19} C_VEL
LIN {X 0,Y 116.589,Z 841.628,A -85,B 0,C 180,E1 27930.887,E2 27930.887} C_VEL
LIN {X 0,Y 115.055,Z 842.502,A -85,B 0,C 180,E1 27931.546,E2 27931.546} C_VEL
LIN {X 0,Y 103.28,Z 849.112,A -85,B 0,C 180,E1 27938.358,E2 27938.358} C_VEL
LIN {X 0,Y 93.003,Z 854.187,A -85,B 0,C 180,E1 27947.368,E2 27947.368} C_VEL
LIN {X 0,Y 85.443,Z 857.53,A -85,B 0,C 180,E1 27959.011,E2 27959.011} C_VEL
LIN {X 0,Y 82.08,Z 858.982,A -85,B 0,C 180,E1 27972.271,E2 27972.271} C_VEL
LIN {X 0,Y 83.032,Z 858.585,A -85,B 0,C 180,E1 27985.166,E2 27985.166} C_VEL
LIN {X 0,Y 84.155,Z 857.882,A -85,B 0,C 180,E1 27990.001,E2 27990.001} C_VEL
LIN {X 0,Y 82.296,Z 854.293,A -85,B 0,C 180,E1 28000.502,E2 28000.502} C_VEL
LIN {X 0,Y 82.921,Z 848.701,A -85,B 0,C 180,E1 28011.951,E2 28011.951} C_VEL
LIN {X 0,Y 86.535,Z 841.109,A -85,B 0,C 180,E1 28022.893,E2 28022.893} C_VEL
LIN {X 0,Y 92.476,Z 831.957,A -85,B 0,C 180,E1 28032.096,E2 28032.096} C_VEL
LIN {X 0,Y 99.867,Z 821.326,A -85,B 0,C 180,E1 28039.545,E2 28039.545} C_VEL
LIN {X 0,Y 108.077,Z 809.228,A -85,B 0,C 180,E1 28045.426,E2 28045.426} C_VEL
LIN {X 0,Y 116.529,Z 795.42,A -85,B 0,C 180,E1 28050.07,E2 28050.07} C_VEL
LIN {X 0,Y 124.509,Z 780.581,A -85,B 0,C 180,E1 28053.561,E2 28053.561} C_VEL
LIN {X 0,Y 131.557,Z 765.099,A -85,B 0,C 180,E1 28056.122,E2 28056.122} C_VEL
LIN {X 0,Y 137.715,Z 748.166,A -85,B 0,C 180,E1 28058.052,E2 28058.052} C_VEL
LIN {X 0,Y 142.513,Z 730.366,A -85,B 0,C 180,E1 28059.461,E2 28059.461} C_VEL
LIN {X 0,Y 145.63,Z 712.55,A -85,B 0,C 180,E1 28060.411,E2 28060.411} C_VEL
LIN {X 0,Y 155.618,Z 608.895,A -85,B 0,C 180,E1 28063.675,E2 28063.675} C_VEL
LIN {X 0,Y 151.692,Z 599.101,A -85,B 0,C 180,E1 28067.351,E2 28067.351} C_VEL
LIN {X 0,Y 147.664,Z 590.432,A -85,B 0,C 180,E1 28071.728,E2 28071.728} C_VEL
LIN {X 0,Y 144.928,Z 585.182,A -85,B 0,C 180,E1 28075.252,E2 28075.252} C_VEL
LIN {X 0,Y 142.674,Z 581.138,A -85,B 0,C 180,E1 28078.796,E2 28078.796} C_VEL
LIN {X 0,Y 140.683,Z 577.6,A -85,B 0,C 180,E1 28082.852,E2 28082.852} C_VEL
LIN {X 0,Y 138.835,Z 574.884,A -85,B 0,C 180,E1 28088.282,E2 28088.282} C_VEL
LIN {X 0,Y 137.98,Z 574.085,A -85,B 0,C 180,E1 28095.123,E2 28095.123} C_VEL
LIN {X 0,Y 138.281,Z 574.848,A -85,B 0,C 180,E1 28099.868,E2 28099.868} C_VEL
LIN {X 0,Y 140.005,Z 578.372,A -85,B 0,C 180,E1 28106.511,E2 28106.511} C_VEL
LIN {X 0,Y 142.927,Z 584.549,A -85,B 0,C 180,E1 28112.724,E2 28112.724} C_VEL
LIN {X 0,Y 145.816,Z 591.225,A -85,B 0,C 180,E1 28117.116,E2 28117.116} C_VEL
LIN {X 0,Y 148.923,Z 598.799,A -85,B 0,C 180,E1 28120.955,E2 28120.955} C_VEL
LIN {X 0,Y 152.008,Z 607.714,A -85,B 0,C 180,E1 28124.338,E2 28124.338} C_VEL
LIN {X 0,Y 151.94,Z 622.951,A -85,B 0,C 180,E1 28125.818,E2 28125.818} C_VEL
LIN {X 0,Y 144,Z 701.493,A -85,B 0,C 180,E1 28128.429,E2 28128.429} C_VEL
LIN {X 0,Y 140.906,Z 719.073,A -85,B 0,C 180,E1 28129.579,E2 28129.579} C_VEL
LIN {X 0,Y 136.5,Z 735.853,A -85,B 0,C 180,E1 28131.222,E2 28131.222} C_VEL
LIN {X 0,Y 130.908,Z 751.573,A -85,B 0,C 180,E1 28133.433,E2 28133.433} C_VEL
LIN {X 0,Y 124.368,Z 766.37,A -85,B 0,C 180,E1 28136.307,E2 28136.307} C_VEL
LIN {X 0,Y 117.426,Z 779.527,A -85,B 0,C 180,E1 28139.842,E2 28139.842} C_VEL
LIN {X 0,Y 109.468,Z 792.535,A -85,B 0,C 180,E1 28144.725,E2 28144.725} C_VEL
LIN {X 0,Y 102.017,Z 803.516,A -85,B 0,C 180,E1 28150.534,E2 28150.534} C_VEL
LIN {X 0,Y 95.029,Z 813.157,A -85,B 0,C 180,E1 28157.851,E2 28157.851} C_VEL
LIN {X 0,Y 89.257,Z 821.337,A -85,B 0,C 180,E1 28166.788,E2 28166.788} C_VEL
LIN {X 0,Y 85.579,Z 827.587,A -85,B 0,C 180,E1 28176.724,E2 28176.724} C_VEL
LIN {X 0,Y 84.221,Z 832.431,A -85,B 0,C 180,E1 28188.237,E2 28188.237} C_VEL
LIN {X 0,Y 85.652,Z 835.362,A -85,B 0,C 180,E1 28199.358,E2 28199.358} C_VEL
LIN {X 0,Y 89.925,Z 836.614,A -85,B 0,C 180,E1 28210.156,E2 28210.156} C_VEL
LIN {X 0,Y 97.383,Z 836.019,A -85,B 0,C 180,E1 28220.356,E2 28220.356} C_VEL
LIN {X 0,Y 106.705,Z 833.634,A -85,B 0,C 180,E1 28228.504,E2 28228.504} C_VEL
LIN {X 0,Y 117.762,Z 829.269,A -85,B 0,C 180,E1 28235.295,E2 28235.295} C_VEL
LIN {X 0,Y 129.382,Z 823.288,A -85,B 0,C 180,E1 28240.59,E2 28240.59} C_VEL
LIN {X 0,Y 141.29,Z 815.623,A -85,B 0,C 180,E1 28244.82,E2 28244.82} C_VEL
LIN {X 0,Y 153.187,Z 806.203,A -85,B 0,C 180,E1 28248.25,E2 28248.25} C_VEL
LIN {X 0,Y 164.14,Z 795.755,A -85,B 0,C 180,E1 28250.886,E2 28250.886} C_VEL
LIN {X 0,Y 174.275,Z 784.133,A -85,B 0,C 180,E1 28252.993,E2 28252.993} C_VEL
LIN {X 0,Y 183.742,Z 770.855,A -85,B 0,C 180,E1 28254.755,E2 28254.755} C_VEL
LIN {X 0,Y 192.388,Z 755.865,A -85,B 0,C 180,E1 28256.226,E2 28256.226} C_VEL
LIN {X 0,Y 199.188,Z 740.861,A -85,B 0,C 180,E1 28257.322,E2 28257.322} C_VEL
LIN {X 0,Y 204.694,Z 724.439,A -85,B 0,C 180,E1 28258.21,E2 28258.21} C_VEL
LIN {X 0,Y 208.614,Z 707.269,A -85,B 0,C 180,E1 28258.868,E2 28258.868} C_VEL
LIN {X 0,Y 213.279,Z 671.232,A -85,B 0,C 180,E1 28259.694,E2 28259.694} C_VEL
LIN {X 0,Y 214.786,Z 659.031,A -85,B 0,C 180,E1 28259.933,E2 28259.933} C_VEL
LIN {X 0,Y 214.461,Z 656.861,A -85,B 0,C 180,E1 28262.137,E2 28262.137} C_VEL
LIN {X 0,Y 214.404,Z 655.291,A -85,B 0,C 180,E1 28265.888,E2 28265.888} C_VEL
LIN {X 0,Y 214.911,Z 655.938,A -85,B 0,C 180,E1 28269.101,E2 28269.101} C_VEL
LIN {X 0,Y 215.307,Z 657.318,A -85,B 0,C 180,E1 28270.756,E2 28270.756} C_VEL
LIN {X 0,Y 208.486,Z 711.53,A -85,B 0,C 180,E1 28271.822,E2 28271.822} C_VEL
LIN {X 0,Y 204.214,Z 729.955,A -85,B 0,C 180,E1 28272.291,E2 28272.291} C_VEL
LIN {X 0,Y 198.46,Z 746.796,A -85,B 0,C 180,E1 28272.874,E2 28272.874} C_VEL
LIN {X 0,Y 190.878,Z 763.251,A -85,B 0,C 180,E1 28273.668,E2 28273.668} C_VEL
LIN {X 0,Y 181.95,Z 778.622,A -85,B 0,C 180,E1 28274.726,E2 28274.726} C_VEL
LIN {X 0,Y 171.751,Z 792.966,A -85,B 0,C 180,E1 28276.148,E2 28276.148} C_VEL
LIN {X 0,Y 160.824,Z 805.703,A -85,B 0,C 180,E1 28277.972,E2 28277.972} C_VEL
LIN {X 0,Y 148.392,Z 817.912,A -85,B 0,C 180,E1 28280.518,E2 28280.518} C_VEL
LIN {X 0,Y 135.566,Z 828.608,A -85,B 0,C 180,E1 28283.859,E2 28283.859} C_VEL
LIN {X 0,Y 122.6,Z 837.794,A -85,B 0,C 180,E1 28288.264,E2 28288.264} C_VEL
LIN {X 0,Y 115.055,Z 842.502,A -85,B 0,C 180,E1 28291.546,E2 28291.546} C_VEL
LIN {X 0,Y 109.313,Z 845.418,A -85,B 0,C 180,E1 28293.786,E2 28293.786} C_VEL
LIN {X 0,Y 95.477,Z 850.341,A -85,B 0,C 180,E1 28298.356,E2 28298.356} C_VEL
LIN {X 0,Y 89.046,Z 852.413,A -85,B 0,C 180,E1 28301.928,E2 28301.928} C_VEL
LIN {X 0,Y 87.771,Z 852.915,A -85,B 0,C 180,E1 28303.055,E2 28303.055} C_VEL
LIN {X 0,Y 79.228,Z 856.149,A -85,B 0,C 180,E1 28314.515,E2 28314.515} C_VEL
LIN {X 0,Y 74.546,Z 857.672,A -85,B 0,C 180,E1 28328.77,E2 28328.77} C_VEL
LIN {X 0,Y 74.703,Z 857.362,A -85,B 0,C 180,E1 28343.083,E2 28343.083} C_VEL
LIN {X 0,Y 76.094,Z 856.491,A -85,B 0,C 180,E1 28350.001,E2 28350.001} C_VEL
LIN {X 0,Y 74.241,Z 852.468,A -85,B 0,C 180,E1 28362.445,E2 28362.445} C_VEL
LIN {X 0,Y 75.533,Z 846.542,A -85,B 0,C 180,E1 28375.064,E2 28375.064} C_VEL
LIN {X 0,Y 80.112,Z 838.614,A -85,B 0,C 180,E1 28386.806,E2 28386.806} C_VEL
LIN {X 0,Y 87.047,Z 829.126,A -85,B 0,C 180,E1 28396.358,E2 28396.358} C_VEL
LIN {X 0,Y 95.355,Z 818.04,A -85,B 0,C 180,E1 28403.844,E2 28403.844} C_VEL
LIN {X 0,Y 104.332,Z 805.358,A -85,B 0,C 180,E1 28409.601,E2 28409.601} C_VEL
LIN {X 0,Y 113.026,Z 791.623,A -85,B 0,C 180,E1 28413.886,E2 28413.886} C_VEL
LIN {X 0,Y 121.171,Z 776.666,A -85,B 0,C 180,E1 28417.094,E2 28417.094} C_VEL
LIN {X 0,Y 128.18,Z 761.174,A -85,B 0,C 180,E1 28419.402,E2 28419.402} C_VEL
LIN {X 0,Y 134.206,Z 744.528,A -85,B 0,C 180,E1 28421.118,E2 28421.118} C_VEL
LIN {X 0,Y 138.751,Z 727.297,A -85,B 0,C 180,E1 28422.37,E2 28422.37} C_VEL
LIN {X 0,Y 141.732,Z 709.282,A -85,B 0,C 180,E1 28423.227,E2 28423.227} C_VEL
LIN {X 0,Y 151.407,Z 612.135,A -85,B 0,C 180,E1 28426.204,E2 28426.204} C_VEL
LIN {X 0,Y 147.749,Z 602.628,A -85,B 0,C 180,E1 28430.162,E2 28430.162} C_VEL
LIN {X 0,Y 144.21,Z 594.749,A -85,B 0,C 180,E1 28434.63,E2 28434.63} C_VEL
LIN {X 0,Y 141.256,Z 588.919,A -85,B 0,C 180,E1 28439.392,E2 28439.392} C_VEL
LIN {X 0,Y 139.274,Z 585.218,A -85,B 0,C 180,E1 28443.706,E2 28443.706} C_VEL
LIN {X 0,Y 137.708,Z 582.729,A -85,B 0,C 180,E1 28448.771,E2 28448.771} C_VEL
LIN {X 0,Y 136.978,Z 582.033,A -85,B 0,C 180,E1 28455.521,E2 28455.521} C_VEL
LIN {X 0,Y 137.203,Z 582.691,A -85,B 0,C 180,E1 28459.366,E2 28459.366} C_VEL
LIN {X 0,Y 138.711,Z 586.125,A -85,B 0,C 180,E1 28465.856,E2 28465.856} C_VEL
LIN {X 0,Y 141.232,Z 592.112,A -85,B 0,C 180,E1 28471.746,E2 28471.746} C_VEL
LIN {X 0,Y 143.563,Z 598.013,A -85,B 0,C 180,E1 28475.683,E2 28475.683} C_VEL
LIN {X 0,Y 146.319,Z 605.403,A -85,B 0,C 180,E1 28479.459,E2 28479.459} C_VEL
LIN {X 0,Y 148.315,Z 611.879,A -85,B 0,C 180,E1 28481.964,E2 28481.964} C_VEL
LIN {X 0,Y 148.101,Z 623.934,A -85,B 0,C 180,E1 28483.144,E2 28483.144} C_VEL
LIN {X 0,Y 139.924,Z 701.992,A -85,B 0,C 180,E1 28485.657,E2 28485.657} C_VEL
LIN {X 0,Y 136.723,Z 719.524,A -85,B 0,C 180,E1 28486.77,E2 28486.77} C_VEL
LIN {X 0,Y 132.299,Z 735.831,A -85,B 0,C 180,E1 28488.311,E2 28488.311} C_VEL
LIN {X 0,Y 126.458,Z 751.765,A -85,B 0,C 180,E1 28490.468,E2 28490.468} C_VEL
LIN {X 0,Y 119.597,Z 766.682,A -85,B 0,C 180,E1 28493.289,E2 28493.289} C_VEL
LIN {X 0,Y 111.919,Z 780.554,A -85,B 0,C 180,E1 28496.977,E2 28496.977} C_VEL
LIN {X 0,Y 103.661,Z 793.307,A -85,B 0,C 180,E1 28501.794,E2 28501.794} C_VEL
LIN {X 0,Y 95.537,Z 804.535,A -85,B 0,C 180,E1 28507.865,E2 28507.865} C_VEL
LIN {X 0,Y 88.006,Z 814.186,A -85,B 0,C 180,E1 28515.524,E2 28515.524} C_VEL
LIN {X 0,Y 81.729,Z 822.383,A -85,B 0,C 180,E1 28525.086,E2 28525.086} C_VEL
LIN {X 0,Y 77.719,Z 828.656,A -85,B 0,C 180,E1 28535.906,E2 28535.906} C_VEL
LIN {X 0,Y 76.281,Z 833.448,A -85,B 0,C 180,E1 28548.334,E2 28548.334} C_VEL
LIN {X 0,Y 77.979,Z 836.501,A -85,B 0,C 180,E1 28560.855,E2 28560.855} C_VEL
LIN {X 0,Y 82.852,Z 837.811,A -85,B 0,C 180,E1 28572.594,E2 28572.594} C_VEL
LIN {X 0,Y 91.055,Z 837.267,A -85,B 0,C 180,E1 28583.282,E2 28583.282} C_VEL
LIN {X 0,Y 101.285,Z 834.911,A -85,B 0,C 180,E1 28591.714,E2 28591.714} C_VEL
LIN {X 0,Y 112.917,Z 830.669,A -85,B 0,C 180,E1 28598.394,E2 28598.394} C_VEL
LIN {X 0,Y 125.096,Z 824.792,A -85,B 0,C 180,E1 28603.56,E2 28603.56} C_VEL
LIN {X 0,Y 137.206,Z 817.466,A -85,B 0,C 180,E1 28607.55,E2 28607.55} C_VEL
LIN {X 0,Y 149.104,Z 808.586,A -85,B 0,C 180,E1 28610.738,E2 28610.738} C_VEL
LIN {X 0,Y 161.045,Z 797.763,A -85,B 0,C 180,E1 28613.396,E2 28613.396} C_VEL
LIN {X 0,Y 171.782,Z 785.993,A -85,B 0,C 180,E1 28615.437,E2 28615.437} C_VEL
LIN {X 0,Y 181.703,Z 772.68,A -85,B 0,C 180,E1 28617.116,E2 28617.116} C_VEL
LIN {X 0,Y 190.602,Z 757.786,A -85,B 0,C 180,E1 28618.496,E2 28618.496} C_VEL
LIN {X 0,Y 197.976,Z 742.077,A -85,B 0,C 180,E1 28619.577,E2 28619.577} C_VEL
LIN {X 0,Y 203.662,Z 725.626,A -85,B 0,C 180,E1 28620.412,E2 28620.412} C_VEL
LIN {X 0,Y 207.764,Z 708.173,A -85,B 0,C 180,E1 28621.044,E2 28621.044} C_VEL
LIN {X 0,Y 212.136,Z 675.399,A -85,B 0,C 180,E1 28621.767,E2 28621.767} C_VEL
LIN {X 0,Y 213.436,Z 664.977,A -85,B 0,C 180,E1 28622.013,E2 28622.013} C_VEL
LIN {X 0,Y 213.383,Z 663.228,A -85,B 0,C 180,E1 28625.916,E2 28625.916} C_VEL
LIN {X 0,Y 213.805,Z 663.744,A -85,B 0,C 180,E1 28628.735,E2 28628.735} C_VEL
LIN {X 0,Y 207.669,Z 711.063,A -85,B 0,C 180,E1 28629.62,E2 28629.62} C_VEL
LIN {X 0,Y 203.338,Z 729.342,A -85,B 0,C 180,E1 28630.04,E2 28630.04} C_VEL
LIN {X 0,Y 197.801,Z 745.345,A -85,B 0,C 180,E1 28630.528,E2 28630.528} C_VEL
LIN {X 0,Y 190.237,Z 761.674,A -85,B 0,C 180,E1 28631.213,E2 28631.213} C_VEL
LIN {X 0,Y 181.031,Z 777.325,A -85,B 0,C 180,E1 28632.153,E2 28632.153} C_VEL
LIN {X 0,Y 170.629,Z 791.731,A -85,B 0,C 180,E1 28633.413,E2 28633.413} C_VEL
LIN {X 0,Y 159.443,Z 804.508,A -85,B 0,C 180,E1 28635.047,E2 28635.047} C_VEL
LIN {X 0,Y 146.65,Z 816.738,A -85,B 0,C 180,E1 28637.348,E2 28637.348} C_VEL
LIN {X 0,Y 133.351,Z 827.441,A -85,B 0,C 180,E1 28640.408,E2 28640.408} C_VEL
LIN {X 0,Y 119.773,Z 836.618,A -85,B 0,C 180,E1 28644.506,E2 28644.506} C_VEL
LIN {X 0,Y 106.337,Z 844.253,A -85,B 0,C 180,E1 28650.114,E2 28650.114} C_VEL
LIN {X 0,Y 93.725,Z 850.362,A -85,B 0,C 180,E1 28657.869,E2 28657.869} C_VEL
LIN {X 0,Y 87.771,Z 852.915,A -85,B 0,C 180,E1 28663.055,E2 28663.055} C_VEL
LIN {X 0,Y 83.031,Z 854.382,A -85,B 0,C 180,E1 28667.066,E2 28667.066} C_VEL
LIN {X 0,Y 71.899,Z 855.971,A -85,B 0,C 180,E1 28676.325,E2 28676.325} C_VEL
LIN {X 0,Y 67.834,Z 856.311,A -85,B 0,C 180,E1 28682.824,E2 28682.824} C_VEL
LIN {X 0,Y 67.301,Z 856.365,A -85,B 0,C 180,E1 28684.654,E2 28684.654} C_VEL
LIN {X 0,Y 66.55,Z 856.066,A -85,B 0,C 180,E1 28701.361,E2 28701.361} C_VEL
LIN {X 0,Y 68.017,Z 855.074,A -85,B 0,C 180,E1 28710.002,E2 28710.002} C_VEL
LIN {X 0,Y 66.279,Z 850.851,A -85,B 0,C 180,E1 28723.969,E2 28723.969} C_VEL
LIN {X 0,Y 68.165,Z 844.759,A -85,B 0,C 180,E1 28737.996,E2 28737.996} C_VEL
LIN {X 0,Y 73.668,Z 836.658,A -85,B 0,C 180,E1 28750.655,E2 28750.655} C_VEL
LIN {X 0,Y 81.141,Z 827.439,A -85,B 0,C 180,E1 28760.152,E2 28760.152} C_VEL
LIN {X 0,Y 90.021,Z 816.44,A -85,B 0,C 180,E1 28767.581,E2 28767.581} C_VEL
LIN {X 0,Y 99.625,Z 803.638,A -85,B 0,C 180,E1 28773.284,E2 28773.284} C_VEL
LIN {X 0,Y 108.816,Z 789.744,A -85,B 0,C 180,E1 28777.437,E2 28777.437} C_VEL
LIN {X 0,Y 117.058,Z 775.056,A -85,B 0,C 180,E1 28780.406,E2 28780.406} C_VEL
LIN {X 0,Y 124.638,Z 758.677,A -85,B 0,C 180,E1 28782.677,E2 28782.677} C_VEL
LIN {X 0,Y 130.651,Z 742.217,A -85,B 0,C 180,E1 28784.232,E2 28784.232} C_VEL
LIN {X 0,Y 135.145,Z 724.92,A -85,B 0,C 180,E1 28785.378,E2 28785.378} C_VEL
LIN {X 0,Y 138.152,Z 706.359,A -85,B 0,C 180,E1 28786.183,E2 28786.183} C_VEL
LIN {X 0,Y 147.496,Z 615.551,A -85,B 0,C 180,E1 28788.861,E2 28788.861} C_VEL
LIN {X 0,Y 144.279,Z 606.959,A -85,B 0,C 180,E1 28792.835,E2 28792.835} C_VEL
LIN {X 0,Y 141.439,Z 600.29,A -85,B 0,C 180,E1 28797.063,E2 28797.063} C_VEL
LIN {X 0,Y 139.543,Z 596.174,A -85,B 0,C 180,E1 28800.617,E2 28800.617} C_VEL
LIN {X 0,Y 137.819,Z 592.723,A -85,B 0,C 180,E1 28804.787,E2 28804.787} C_VEL
LIN {X 0,Y 136.593,Z 590.575,A -85,B 0,C 180,E1 28809.268,E2 28809.268} C_VEL
LIN {X 0,Y 135.978,Z 589.984,A -85,B 0,C 180,E1 28815.788,E2 28815.788} C_VEL
LIN {X 0,Y 136.154,Z 590.643,A -85,B 0,C 180,E1 28819.075,E2 28819.075} C_VEL
LIN {X 0,Y 137.434,Z 593.883,A -85,B 0,C 180,E1 28825.19,E2 28825.19} C_VEL
LIN {X 0,Y 139.57,Z 599.623,A -85,B 0,C 180,E1 28830.72,E2 28830.72} C_VEL
LIN {X 0,Y 141.488,Z 605.052,A -85,B 0,C 180,E1 28834.352,E2 28834.352} C_VEL
LIN {X 0,Y 144.015,Z 612.72,A -85,B 0,C 180,E1 28838.234,E2 28838.234} C_VEL
LIN {X 0,Y 144.875,Z 616.073,A -85,B 0,C 180,E1 28839.481,E2 28839.481} C_VEL
LIN {X 0,Y 144.58,Z 625.114,A -85,B 0,C 180,E1 28840.34,E2 28840.34} C_VEL
LIN {X 0,Y 136.169,Z 702.656,A -85,B 0,C 180,E1 28842.733,E2 28842.733} C_VEL
LIN {X 0,Y 132.835,Z 720.19,A -85,B 0,C 180,E1 28843.807,E2 28843.807} C_VEL
LIN {X 0,Y 128.054,Z 737.071,A -85,B 0,C 180,E1 28845.353,E2 28845.353} C_VEL
LIN {X 0,Y 121.965,Z 752.877,A -85,B 0,C 180,E1 28847.441,E2 28847.441} C_VEL
LIN {X 0,Y 114.792,Z 767.746,A -85,B 0,C 180,E1 28850.192,E2 28850.192} C_VEL
LIN {X 0,Y 107.099,Z 781.006,A -85,B 0,C 180,E1 28853.641,E2 28853.641} C_VEL
LIN {X 0,Y 98.682,Z 793.358,A -85,B 0,C 180,E1 28858.204,E2 28858.204} C_VEL
LIN {X 0,Y 89.816,Z 804.885,A -85,B 0,C 180,E1 28864.388,E2 28864.388} C_VEL
LIN {X 0,Y 81.685,Z 814.595,A -85,B 0,C 180,E1 28872.18,E2 28872.18} C_VEL
LIN {X 0,Y 74.66,Z 822.934,A -85,B 0,C 180,E1 28882.326,E2 28882.326} C_VEL
LIN {X 0,Y 70.08,Z 829.351,A -85,B 0,C 180,E1 28894.089,E2 28894.089} C_VEL
LIN {X 0,Y 68.337,Z 834.327,A -85,B 0,C 180,E1 28907.999,E2 28907.999} C_VEL
LIN {X 0,Y 70.369,Z 837.634,A -85,B 0,C 180,E1 28922.677,E2 28922.677} C_VEL
LIN {X 0,Y 75.881,Z 839.006,A -85,B 0,C 180,E1 28935.359,E2 28935.359} C_VEL
LIN {X 0,Y 84.611,Z 838.567,A -85,B 0,C 180,E1 28946.26,E2 28946.26} C_VEL
LIN {X 0,Y 95.912,Z 836.255,A -85,B 0,C 180,E1 28955.085,E2 28955.085} C_VEL
LIN {X 0,Y 108.31,Z 832.119,A -85,B 0,C 180,E1 28961.706,E2 28961.706} C_VEL
LIN {X 0,Y 121.21,Z 826.272,A -85,B 0,C 180,E1 28966.746,E2 28966.746} C_VEL
LIN {X 0,Y 133.8,Z 819.061,A -85,B 0,C 180,E1 28970.538,E2 28970.538} C_VEL
LIN {X 0,Y 145.918,Z 810.522,A -85,B 0,C 180,E1 28973.491,E2 28973.491} C_VEL
LIN {X 0,Y 158.36,Z 799.733,A -85,B 0,C 180,E1 28976.01,E2 28976.01} C_VEL
LIN {X 0,Y 170.076,Z 787.334,A -85,B 0,C 180,E1 28978.021,E2 28978.021} C_VEL
LIN {X 0,Y 179.979,Z 774.505,A -85,B 0,C 180,E1 28979.526,E2 28979.526} C_VEL
LIN {X 0,Y 188.99,Z 759.946,A -85,B 0,C 180,E1 28980.788,E2 28980.788} C_VEL
LIN {X 0,Y 196.566,Z 744.43,A -85,B 0,C 180,E1 28981.792,E2 28981.792} C_VEL
LIN {X 0,Y 202.331,Z 728.869,A -85,B 0,C 180,E1 28982.549,E2 28982.549} C_VEL
LIN {X 0,Y 206.657,Z 711.948,A -85,B 0,C 180,E1 28983.151,E2 28983.151} C_VEL
LIN {X 0,Y 209.987,Z 689.663,A -85,B 0,C 180,E1 28983.681,E2 28983.681} C_VEL
LIN {X 0,Y 212.245,Z 671.938,A -85,B 0,C 180,E1 28984.052,E2 28984.052} C_VEL
LIN {X 0,Y 212.388,Z 671.179,A -85,B 0,C 180,E1 28986.215,E2 28986.215} C_VEL
LIN {X 0,Y 212.429,Z 671.323,A -85,B 0,C 180,E1 28986.723,E2 28986.723} C_VEL
LIN {X 0,Y 207.128,Z 710.773,A -85,B 0,C 180,E1 28987.406,E2 28987.406} C_VEL
LIN {X 0,Y 202.772,Z 728.788,A -85,B 0,C 180,E1 28987.775,E2 28987.775} C_VEL
LIN {X 0,Y 196.99,Z 745.162,A -85,B 0,C 180,E1 28988.21,E2 28988.21} C_VEL
LIN {X 0,Y 189.203,Z 761.565,A -85,B 0,C 180,E1 28988.808,E2 28988.808} C_VEL
LIN {X 0,Y 180.048,Z 776.804,A -85,B 0,C 180,E1 28989.606,E2 28989.606} C_VEL
LIN {X 0,Y 169.425,Z 791.146,A -85,B 0,C 180,E1 28990.707,E2 28990.707} C_VEL
LIN {X 0,Y 157.541,Z 804.276,A -85,B 0,C 180,E1 28992.212,E2 28992.212} C_VEL
LIN {X 0,Y 144.441,Z 816.354,A -85,B 0,C 180,E1 28994.279,E2 28994.279} C_VEL
LIN {X 0,Y 130.736,Z 826.928,A -85,B 0,C 180,E1 28997.064,E2 28997.064} C_VEL
LIN {X 0,Y 116.623,Z 835.935,A -85,B 0,C 180,E1 29000.854,E2 29000.854} C_VEL
LIN {X 0,Y 102.47,Z 843.458,A -85,B 0,C 180,E1 29006.145,E2 29006.145} C_VEL
LIN {X 0,Y 88.921,Z 849.443,A -85,B 0,C 180,E1 29013.689,E2 29013.689} C_VEL
LIN {X 0,Y 77.604,Z 853.515,A -85,B 0,C 180,E1 29023.822,E2 29023.822} C_VEL
LIN {X 0,Y 69.349,Z 855.913,A -85,B 0,C 180,E1 29037.762,E2 29037.762} C_VEL
LIN {X 0,Y 67.301,Z 856.365,A -85,B 0,C 180,E1 29044.654,E2 29044.654} C_VEL
LIN {X 0,Y 65.373,Z 856.314,A -85,B 0,C 180,E1 29051.699,E2 29051.699} C_VEL
LIN {X 0,Y 62.581,Z 855.458,A -85,B 0,C 180,E1 29060.365,E2 29060.365} C_VEL
LIN {X 0,Y 59.492,Z 853.176,A -85,B 0,C 180,E1 29072.116,E2 29072.116} C_VEL
LIN {X 0,Y 58.821,Z 852.067,A -85,B 0,C 180,E1 29076.344,E2 29076.344} C_VEL
LIN {X 0,Y 59.002,Z 846.732,A -85,B 0,C 180,E1 29092.942,E2 29092.942} C_VEL
LIN {X 0,Y 63.568,Z 839.47,A -85,B 0,C 180,E1 29108.148,E2 29108.148} C_VEL
LIN {X 0,Y 70.931,Z 830.963,A -85,B 0,C 180,E1 29119.579,E2 29119.579} C_VEL
LIN {X 0,Y 79.999,Z 820.795,A -85,B 0,C 180,E1 29128.202,E2 29128.202} C_VEL
LIN {X 0,Y 90.14,Z 808.712,A -85,B 0,C 180,E1 29134.695,E2 29134.695} C_VEL
LIN {X 0,Y 100.137,Z 795.271,A -85,B 0,C 180,E1 29139.383,E2 29139.383} C_VEL
LIN {X 0,Y 108.977,Z 781.348,A -85,B 0,C 180,E1 29142.595,E2 29142.595} C_VEL
LIN {X 0,Y 116.992,Z 766.245,A -85,B 0,C 180,E1 29144.963,E2 29144.963} C_VEL
LIN {X 0,Y 123.82,Z 750.334,A -85,B 0,C 180,E1 29146.672,E2 29146.672} C_VEL
LIN {X 0,Y 129.333,Z 733.398,A -85,B 0,C 180,E1 29147.935,E2 29147.935} C_VEL
LIN {X 0,Y 133.216,Z 715.622,A -85,B 0,C 180,E1 29148.852,E2 29148.852} C_VEL
LIN {X 0,Y 136.406,Z 689.317,A -85,B 0,C 180,E1 29149.687,E2 29149.687} C_VEL
LIN {X 0,Y 143.84,Z 619.105,A -85,B 0,C 180,E1 29151.657,E2 29151.657} C_VEL
LIN {X 0,Y 141.125,Z 611.375,A -85,B 0,C 180,E1 29155.633,E2 29155.633} C_VEL
LIN {X 0,Y 138.836,Z 605.536,A -85,B 0,C 180,E1 29159.795,E2 29159.795} C_VEL
LIN {X 0,Y 136.697,Z 600.681,A -85,B 0,C 180,E1 29165.036,E2 29165.036} C_VEL
LIN {X 0,Y 135.488,Z 598.425,A -85,B 0,C 180,E1 29169.773,E2 29169.773} C_VEL
LIN {X 0,Y 134.98,Z 597.931,A -85,B 0,C 180,E1 29175.908,E2 29175.908} C_VEL
LIN {X 0,Y 135.102,Z 598.545,A -85,B 0,C 180,E1 29178.682,E2 29178.682} C_VEL
LIN {X 0,Y 136.146,Z 601.562,A -85,B 0,C 180,E1 29184.402,E2 29184.402} C_VEL
LIN {X 0,Y 137.903,Z 606.951,A -85,B 0,C 180,E1 29189.541,E2 29189.541} C_VEL
LIN {X 0,Y 139.508,Z 612.134,A -85,B 0,C 180,E1 29193.012,E2 29193.012} C_VEL
LIN {X 0,Y 141.674,Z 619.63,A -85,B 0,C 180,E1 29196.799,E2 29196.799} C_VEL
LIN {X 0,Y 141.389,Z 625.979,A -85,B 0,C 180,E1 29197.405,E2 29197.405} C_VEL
LIN {X 0,Y 132.754,Z 703.146,A -85,B 0,C 180,E1 29199.656,E2 29199.656} C_VEL
LIN {X 0,Y 129.318,Z 720.646,A -85,B 0,C 180,E1 29200.672,E2 29200.672} C_VEL
LIN {X 0,Y 124.59,Z 736.875,A -85,B 0,C 180,E1 29202.068,E2 29202.068} C_VEL
LIN {X 0,Y 118.665,Z 752.061,A -85,B 0,C 180,E1 29203.92,E2 29203.92} C_VEL
LIN {X 0,Y 111.168,Z 767.206,A -85,B 0,C 180,E1 29206.523,E2 29206.523} C_VEL
LIN {X 0,Y 102.668,Z 781.364,A -85,B 0,C 180,E1 29210.001,E2 29210.001} C_VEL
LIN {X 0,Y 94.126,Z 793.343,A -85,B 0,C 180,E1 29214.249,E2 29214.249} C_VEL
LIN {X 0,Y 84.701,Z 804.9,A -85,B 0,C 180,E1 29220.276,E2 29220.276} C_VEL
LIN {X 0,Y 75.685,Z 814.967,A -85,B 0,C 180,E1 29228.289,E2 29228.289} C_VEL
LIN {X 0,Y 67.826,Z 823.436,A -85,B 0,C 180,E1 29238.95,E2 29238.95} C_VEL
LIN {X 0,Y 62.279,Z 830.392,A -85,B 0,C 180,E1 29252.759,E2 29252.759} C_VEL
LIN {X 0,Y 60.397,Z 835.142,A -85,B 0,C 180,E1 29267.335,E2 29267.335} C_VEL
LIN {X 0,Y 62.491,Z 838.566,A -85,B 0,C 180,E1 29283.691,E2 29283.691} C_VEL
LIN {X 0,Y 68.667,Z 840.151,A -85,B 0,C 180,E1 29297.952,E2 29297.952} C_VEL
LIN {X 0,Y 77.941,Z 839.927,A -85,B 0,C 180,E1 29309.259,E2 29309.259} C_VEL
LIN {X 0,Y 89.504,Z 837.92,A -85,B 0,C 180,E1 29318,E2 29318} C_VEL
LIN {X 0,Y 102.864,Z 834.023,A -85,B 0,C 180,E1 29324.784,E2 29324.784} C_VEL
LIN {X 0,Y 115.917,Z 828.67,A -85,B 0,C 180,E1 29329.563,E2 29329.563} C_VEL
LIN {X 0,Y 129.83,Z 821.245,A -85,B 0,C 180,E1 29333.44,E2 29333.44} C_VEL
LIN {X 0,Y 143.261,Z 812.272,A -85,B 0,C 180,E1 29336.4,E2 29336.4} C_VEL
LIN {X 0,Y 156.016,Z 801.703,A -85,B 0,C 180,E1 29338.709,E2 29338.709} C_VEL
LIN {X 0,Y 167.982,Z 789.503,A -85,B 0,C 180,E1 29340.547,E2 29340.547} C_VEL
LIN {X 0,Y 178.529,Z 776.341,A -85,B 0,C 180,E1 29341.975,E2 29341.975} C_VEL
LIN {X 0,Y 187.75,Z 761.988,A -85,B 0,C 180,E1 29343.123,E2 29343.123} C_VEL
LIN {X 0,Y 195.455,Z 746.782,A -85,B 0,C 180,E1 29344.035,E2 29344.035} C_VEL
LIN {X 0,Y 201.666,Z 730.74,A -85,B 0,C 180,E1 29344.762,E2 29344.762} C_VEL
LIN {X 0,Y 205.78,Z 715.945,A -85,B 0,C 180,E1 29345.278,E2 29345.278} C_VEL
LIN {X 0,Y 200.93,Z 733.162,A -85,B 0,C 180,E1 29345.601,E2 29345.601} C_VEL
LIN {X 0,Y 194.494,Z 749.515,A -85,B 0,C 180,E1 29346,E2 29346} C_VEL
LIN {X 0,Y 186.675,Z 764.784,A -85,B 0,C 180,E1 29346.507,E2 29346.507} C_VEL
LIN {X 0,Y 176.801,Z 780.003,A -85,B 0,C 180,E1 29347.245,E2 29347.245} C_VEL
LIN {X 0,Y 165.692,Z 793.939,A -85,B 0,C 180,E1 29348.255,E2 29348.255} C_VEL
LIN {X 0,Y 153.154,Z 806.904,A -85,B 0,C 180,E1 29349.672,E2 29349.672} C_VEL
LIN {X 0,Y 139.821,Z 818.245,A -85,B 0,C 180,E1 29351.571,E2 29351.571} C_VEL
LIN {X 0,Y 124.872,Z 828.788,A -85,B 0,C 180,E1 29354.371,E2 29354.371} C_VEL
LIN {X 0,Y 110.405,Z 837.211,A -85,B 0,C 180,E1 29358.029,E2 29358.029} C_VEL
LIN {X 0,Y 95.783,Z 844.128,A -85,B 0,C 180,E1 29363.279,E2 29363.279} C_VEL
LIN {X 0,Y 81.657,Z 849.513,A -85,B 0,C 180,E1 29371.008,E2 29371.008} C_VEL
LIN {X 0,Y 69.775,Z 853.088,A -85,B 0,C 180,E1 29381.831,E2 29381.831} C_VEL
LIN {X 0,Y 61.496,Z 854.935,A -85,B 0,C 180,E1 29396.443,E2 29396.443} C_VEL
LIN {X 0,Y 58.306,Z 854.979,A -85,B 0,C 180,E1 29415.096,E2 29415.096} C_VEL
LIN {X 0,Y 59.99,Z 853.671,A -85,B 0,C 180,E1 29429.723,E2 29429.723} C_VEL
LIN {X 0,Y 58.821,Z 852.067,A -85,B 0,C 180,E1 29436.344,E2 29436.344} C_VEL
LIN {X 0,Y 57.358,Z 849.888,A -85,B 0,C 180,E1 29443.537,E2 29443.537} C_VEL
LIN {X 0,Y 54.154,Z 844.433,A -85,B 0,C 180,E1 29458.362,E2 29458.362} C_VEL
LIN {X 0,Y 54.669,Z 840.836,A -85,B 0,C 180,E1 29466.973,E2 29466.973} C_VEL
LIN {X 0,Y 55.678,Z 839.367,A -85,B 0,C 180,E1 29469.931,E2 29469.931} C_VEL
LIN {X 0,Y 63.924,Z 830.778,A -85,B 0,C 180,E1 29482.914,E2 29482.914} C_VEL
LIN {X 0,Y 73.674,Z 820.868,A -85,B 0,C 180,E1 29491.905,E2 29491.905} C_VEL
LIN {X 0,Y 83.999,Z 809.483,A -85,B 0,C 180,E1 29498.198,E2 29498.198} C_VEL
LIN {X 0,Y 94.679,Z 796.049,A -85,B 0,C 180,E1 29502.891,E2 29502.891} C_VEL
LIN {X 0,Y 104.064,Z 782.223,A -85,B 0,C 180,E1 29506.034,E2 29506.034} C_VEL
LIN {X 0,Y 112.336,Z 767.545,A -85,B 0,C 180,E1 29508.26,E2 29508.26} C_VEL
LIN {X 0,Y 119.827,Z 750.986,A -85,B 0,C 180,E1 29509.943,E2 29509.943} C_VEL
LIN {X 0,Y 125.497,Z 734.544,A -85,B 0,C 180,E1 29511.096,E2 29511.096} C_VEL
LIN {X 0,Y 129.632,Z 717.2,A -85,B 0,C 180,E1 29511.965,E2 29511.965} C_VEL
LIN {X 0,Y 132.528,Z 695.876,A -85,B 0,C 180,E1 29512.635,E2 29512.635} C_VEL
LIN {X 0,Y 140.563,Z 623.01,A -85,B 0,C 180,E1 29514.49,E2 29514.49} C_VEL
LIN {X 0,Y 138.295,Z 615.99,A -85,B 0,C 180,E1 29518.551,E2 29518.551} C_VEL
LIN {X 0,Y 136.449,Z 611.029,A -85,B 0,C 180,E1 29522.731,E2 29522.731} C_VEL
LIN {X 0,Y 135.179,Z 607.957,A -85,B 0,C 180,E1 29526.584,E2 29526.584} C_VEL
LIN {X 0,Y 134.391,Z 606.277,A -85,B 0,C 180,E1 29530.287,E2 29530.287} C_VEL
LIN {X 0,Y 133.99,Z 605.918,A -85,B 0,C 180,E1 29536.474,E2 29536.474} C_VEL
LIN {X 0,Y 134.379,Z 607.797,A -85,B 0,C 180,E1 29541.155,E2 29541.155} C_VEL
LIN {X 0,Y 134.973,Z 609.744,A -85,B 0,C 180,E1 29544.045,E2 29544.045} C_VEL
LIN {X 0,Y 136.241,Z 614.063,A -85,B 0,C 180,E1 29548.17,E2 29548.17} C_VEL
LIN {X 0,Y 137.738,Z 619.654,A -85,B 0,C 180,E1 29551.914,E2 29551.914} C_VEL
LIN {X 0,Y 138.78,Z 624.288,A -85,B 0,C 180,E1 29554.165,E2 29554.165} C_VEL
LIN {X 0,Y 137.94,Z 632.465,A -85,B 0,C 180,E1 29554.478,E2 29554.478} C_VEL
LIN {X 0,Y 129.688,Z 703.922,A -85,B 0,C 180,E1 29556.44,E2 29556.44} C_VEL
LIN {X 0,Y 126.099,Z 721.498,A -85,B 0,C 180,E1 29557.4,E2 29557.4} C_VEL
LIN {X 0,Y 121.119,Z 737.938,A -85,B 0,C 180,E1 29558.727,E2 29558.727} C_VEL
LIN {X 0,Y 114.544,Z 753.938,A -85,B 0,C 180,E1 29560.585,E2 29560.585} C_VEL
LIN {X 0,Y 106.739,Z 768.919,A -85,B 0,C 180,E1 29563.057,E2 29563.057} C_VEL
LIN {X 0,Y 97.851,Z 782.901,A -85,B 0,C 180,E1 29566.39,E2 29566.39} C_VEL
LIN {X 0,Y 88.456,Z 795.259,A -85,B 0,C 180,E1 29570.727,E2 29570.727} C_VEL
LIN {X 0,Y 78.467,Z 806.669,A -85,B 0,C 180,E1 29576.773,E2 29576.773} C_VEL
LIN {X 0,Y 68.79,Z 816.566,A -85,B 0,C 180,E1 29585.068,E2 29585.068} C_VEL
LIN {X 0,Y 60.264,Z 824.942,A -85,B 0,C 180,E1 29596.567,E2 29596.567} C_VEL
LIN {X 0,Y 54.52,Z 831.433,A -85,B 0,C 180,E1 29611.049,E2 29611.049} C_VEL
LIN {X 0,Y 52.451,Z 836.232,A -85,B 0,C 180,E1 29627.756,E2 29627.756} C_VEL
LIN {X 0,Y 54.826,Z 839.593,A -85,B 0,C 180,E1 29645.701,E2 29645.701} C_VEL
LIN {X 0,Y 62.174,Z 841.326,A -85,B 0,C 180,E1 29661.997,E2 29661.997} C_VEL
LIN {X 0,Y 72.787,Z 841.143,A -85,B 0,C 180,E1 29673.921,E2 29673.921} C_VEL
LIN {X 0,Y 85.85,Z 839.054,A -85,B 0,C 180,E1 29682.747,E2 29682.747} C_VEL
LIN {X 0,Y 99.971,Z 835.16,A -85,B 0,C 180,E1 29689.044,E2 29689.044} C_VEL
LIN {X 0,Y 113.726,Z 829.746,A -85,B 0,C 180,E1 29693.443,E2 29693.443} C_VEL
LIN {X 0,Y 128.163,Z 822.297,A -85,B 0,C 180,E1 29696.939,E2 29696.939} C_VEL
LIN {X 0,Y 142.06,Z 813.259,A -85,B 0,C 180,E1 29699.596,E2 29699.596} C_VEL
LIN {X 0,Y 155.039,Z 802.738,A -85,B 0,C 180,E1 29701.633,E2 29701.633} C_VEL
LIN {X 0,Y 167.245,Z 790.556,A -85,B 0,C 180,E1 29703.26,E2 29703.26} C_VEL
LIN {X 0,Y 177.879,Z 777.586,A -85,B 0,C 180,E1 29704.534,E2 29704.534} C_VEL
LIN {X 0,Y 166.695,Z 791.686,A -85,B 0,C 180,E1 29705.328,E2 29705.328} C_VEL
LIN {X 0,Y 153.958,Z 804.871,A -85,B 0,C 180,E1 29706.472,E2 29706.472} C_VEL
LIN {X 0,Y 140.354,Z 816.41,A -85,B 0,C 180,E1 29708.028,E2 29708.028} C_VEL
LIN {X 0,Y 125.967,Z 826.457,A -85,B 0,C 180,E1 29710.188,E2 29710.188} C_VEL
LIN {X 0,Y 110.929,Z 835.078,A -85,B 0,C 180,E1 29713.234,E2 29713.234} C_VEL
LIN {X 0,Y 95.461,Z 842.257,A -85,B 0,C 180,E1 29717.682,E2 29717.682} C_VEL
LIN {X 0,Y 80.158,Z 847.797,A -85,B 0,C 180,E1 29724.419,E2 29724.419} C_VEL
LIN {X 0,Y 65.913,Z 851.685,A -85,B 0,C 180,E1 29735.003,E2 29735.003} C_VEL
LIN {X 0,Y 55.702,Z 853.602,A -85,B 0,C 180,E1 29749.747,E2 29749.747} C_VEL
LIN {X 0,Y 50.59,Z 853.723,A -85,B 0,C 180,E1 29770.369,E2 29770.369} C_VEL
LIN {X 0,Y 51.931,Z 852.244,A -85,B 0,C 180,E1 29789.45,E2 29789.45} C_VEL
LIN {X 0,Y 50.53,Z 847.599,A -85,B 0,C 180,E1 29808.46,E2 29808.46} C_VEL
LIN {X 0,Y 54.164,Z 841.19,A -85,B 0,C 180,E1 29826.21,E2 29826.21} C_VEL
LIN {X 0,Y 55.678,Z 839.367,A -85,B 0,C 180,E1 29829.931,E2 29829.931} C_VEL
LIN {X 0,Y 58.013,Z 835.821,A -85,B 0,C 180,E1 29836.474,E2 29836.474} C_VEL
LIN {X 0,Y 61.912,Z 827.926,A -85,B 0,C 180,E1 29848.884,E2 29848.884} C_VEL
LIN {X 0,Y 65.689,Z 822.892,A -85,B 0,C 180,E1 29854.589,E2 29854.589} C_VEL
LIN {X 0,Y 67.628,Z 820.901,A -85,B 0,C 180,E1 29856.214,E2 29856.214} C_VEL
LIN {X 0,Y 78.657,Z 809.721,A -85,B 0,C 180,E1 29862.439,E2 29862.439} C_VEL
LIN {X 0,Y 89.376,Z 797.115,A -85,B 0,C 180,E1 29866.729,E2 29866.729} C_VEL
LIN {X 0,Y 99.563,Z 782.978,A -85,B 0,C 180,E1 29869.796,E2 29869.796} C_VEL
LIN {X 0,Y 108.477,Z 768.043,A -85,B 0,C 180,E1 29871.911,E2 29871.911} C_VEL
LIN {X 0,Y 116.101,Z 751.997,A -85,B 0,C 180,E1 29873.4,E2 29873.4} C_VEL
LIN {X 0,Y 122.3,Z 734.858,A -85,B 0,C 180,E1 29874.489,E2 29874.489} C_VEL
LIN {X 0,Y 126.697,Z 717.378,A -85,B 0,C 180,E1 29875.292,E2 29875.292} C_VEL
LIN {X 0,Y 129.586,Z 697.344,A -85,B 0,C 180,E1 29875.878,E2 29875.878} C_VEL
LIN {X 0,Y 137.549,Z 626.809,A -85,B 0,C 180,E1 29877.605,E2 29877.605} C_VEL
LIN {X 0,Y 135.836,Z 621.062,A -85,B 0,C 180,E1 29881.477,E2 29881.477} C_VEL
LIN {X 0,Y 134.739,Z 617.911,A -85,B 0,C 180,E1 29884.47,E2 29884.47} C_VEL
LIN {X 0,Y 133.856,Z 615.46,A -85,B 0,C 180,E1 29887.728,E2 29887.728} C_VEL
LIN {X 0,Y 133.243,Z 614.047,A -85,B 0,C 180,E1 29891.252,E2 29891.252} C_VEL
LIN {X 0,Y 133.006,Z 613.959,A -85,B 0,C 180,E1 29897.049,E2 29897.049} C_VEL
LIN {X 0,Y 133.58,Z 616.716,A -85,B 0,C 180,E1 29902.442,E2 29902.442} C_VEL
LIN {X 0,Y 134.643,Z 621.232,A -85,B 0,C 180,E1 29906.817,E2 29906.817} C_VEL
LIN {X 0,Y 135.87,Z 626.744,A -85,B 0,C 180,E1 29910.455,E2 29910.455} C_VEL
LIN {X 0,Y 136.106,Z 628.405,A -85,B 0,C 180,E1 29911.182,E2 29911.182} C_VEL
LIN {X 0,Y 127.131,Z 704.202,A -85,B 0,C 180,E1 29913.059,E2 29913.059} C_VEL
LIN {X 0,Y 123.481,Z 721.699,A -85,B 0,C 180,E1 29913.929,E2 29913.929} C_VEL
LIN {X 0,Y 118.535,Z 737.708,A -85,B 0,C 180,E1 29915.093,E2 29915.093} C_VEL
LIN {X 0,Y 112.174,Z 753.105,A -85,B 0,C 180,E1 29916.671,E2 29916.671} C_VEL
LIN {X 0,Y 104.073,Z 768.365,A -85,B 0,C 180,E1 29918.903,E2 29918.903} C_VEL
LIN {X 0,Y 94.596,Z 782.892,A -85,B 0,C 180,E1 29922.01,E2 29922.01} C_VEL
LIN {X 0,Y 84.855,Z 795.241,A -85,B 0,C 180,E1 29925.955,E2 29925.955} C_VEL
LIN {X 0,Y 74.154,Z 806.821,A -85,B 0,C 180,E1 29931.664,E2 29931.664} C_VEL
LIN {X 0,Y 63.569,Z 816.93,A -85,B 0,C 180,E1 29939.778,E2 29939.778} C_VEL
LIN {X 0,Y 53.932,Z 825.455,A -85,B 0,C 180,E1 29951.627,E2 29951.627} C_VEL
LIN {X 0,Y 46.826,Z 832.473,A -85,B 0,C 180,E1 29968.774,E2 29968.774} C_VEL
LIN {X 0,Y 44.522,Z 837.511,A -85,B 0,C 180,E1 29989.392,E2 29989.392} C_VEL
LIN {X 0,Y 47.849,Z 840.871,A -85,B 0,C 180,E1 30010.372,E2 30010.372} C_VEL
LIN {X 0,Y 56.702,Z 842.557,A -85,B 0,C 180,E1 30027.821,E2 30027.821} C_VEL
LIN {X 0,Y 68.509,Z 842.33,A -85,B 0,C 180,E1 30039.494,E2 30039.494} C_VEL
LIN {X 0,Y 82.835,Z 840.19,A -85,B 0,C 180,E1 30047.876,E2 30047.876} C_VEL
LIN {X 0,Y 97.668,Z 836.294,A -85,B 0,C 180,E1 30053.533,E2 30053.533} C_VEL
LIN {X 0,Y 112.093,Z 830.813,A -85,B 0,C 180,E1 30057.457,E2 30057.457} C_VEL
LIN {X 0,Y 126.986,Z 823.35,A -85,B 0,C 180,E1 30060.516,E2 30060.516} C_VEL
LIN {X 0,Y 141.335,Z 814.243,A -85,B 0,C 180,E1 30062.838,E2 30062.838} C_VEL
LIN {X 0,Y 148.696,Z 808.672,A -85,B 0,C 180,E1 30063.855,E2 30063.855} C_VEL
LIN {X 0,Y 134.548,Z 819.587,A -85,B 0,C 180,E1 30065.269,E2 30065.269} C_VEL
LIN {X 0,Y 119.935,Z 828.803,A -85,B 0,C 180,E1 30067.229,E2 30067.229} C_VEL
LIN {X 0,Y 103.64,Z 837.103,A -85,B 0,C 180,E1 30070.256,E2 30070.256} C_VEL
LIN {X 0,Y 87.822,Z 843.461,A -85,B 0,C 180,E1 30074.599,E2 30074.599} C_VEL
LIN {X 0,Y 71.992,Z 848.239,A -85,B 0,C 180,E1 30081.487,E2 30081.487} C_VEL
LIN {X 0,Y 57.209,Z 851.362,A -85,B 0,C 180,E1 30092.978,E2 30092.978} C_VEL
LIN {X 0,Y 46.385,Z 852.605,A -85,B 0,C 180,E1 30111.312,E2 30111.312} C_VEL
LIN {X 0,Y 42.611,Z 851.885,A -85,B 0,C 180,E1 30136.431,E2 30136.431} C_VEL
LIN {X 0,Y 43.805,Z 850.765,A -85,B 0,C 180,E1 30149.348,E2 30149.348} C_VEL
LIN {X 0,Y 42.825,Z 845.964,A -85,B 0,C 180,E1 30171.938,E2 30171.938} C_VEL
LIN {X 0,Y 47.76,Z 839.346,A -85,B 0,C 180,E1 30192.064,E2 30192.064} C_VEL
LIN {X 0,Y 56.508,Z 831.167,A -85,B 0,C 180,E1 30206.27,E2 30206.27} C_VEL
LIN {X 0,Y 67.628,Z 820.901,A -85,B 0,C 180,E1 30216.214,E2 30216.214} C_VEL
LIN {X 0,Y 71.883,Z 816.182,A -85,B 0,C 180,E1 30219.897,E2 30219.897} C_VEL
LIN {X 0,Y 78.798,Z 806.104,A -85,B 0,C 180,E1 30227.385,E2 30227.385} C_VEL
LIN {X 0,Y 83.293,Z 799.78,A -85,B 0,C 180,E1 30230.501,E2 30230.501} C_VEL
LIN {X 0,Y 85.236,Z 797.294,A -85,B 0,C 180,E1 30231.24,E2 30231.24} C_VEL
LIN {X 0,Y 95.53,Z 783.73,A -85,B 0,C 180,E1 30233.894,E2 30233.894} C_VEL
LIN {X 0,Y 104.774,Z 768.991,A -85,B 0,C 180,E1 30235.757,E2 30235.757} C_VEL
LIN {X 0,Y 112.636,Z 753.437,A -85,B 0,C 180,E1 30237.046,E2 30237.046} C_VEL
LIN {X 0,Y 119.059,Z 736.713,A -85,B 0,C 180,E1 30237.977,E2 30237.977} C_VEL
LIN {X 0,Y 123.912,Z 718.78,A -85,B 0,C 180,E1 30238.718,E2 30238.718} C_VEL
LIN {X 0,Y 126.841,Z 700.844,A -85,B 0,C 180,E1 30239.215,E2 30239.215} C_VEL
LIN {X 0,Y 134.969,Z 631.101,A -85,B 0,C 180,E1 30240.715,E2 30240.715} C_VEL
LIN {X 0,Y 133.589,Z 626.055,A -85,B 0,C 180,E1 30244.723,E2 30244.723} C_VEL
LIN {X 0,Y 132.629,Z 623.075,A -85,B 0,C 180,E1 30248.673,E2 30248.673} C_VEL
LIN {X 0,Y 132.176,Z 621.91,A -85,B 0,C 180,E1 30251.786,E2 30251.786} C_VEL
LIN {X 0,Y 131.989,Z 621.904,A -85,B 0,C 180,E1 30256.731,E2 30256.731} C_VEL
LIN {X 0,Y 132.361,Z 624.364,A -85,B 0,C 180,E1 30261.493,E2 30261.493} C_VEL
